KUKA KRL program: MyProgram_321().src

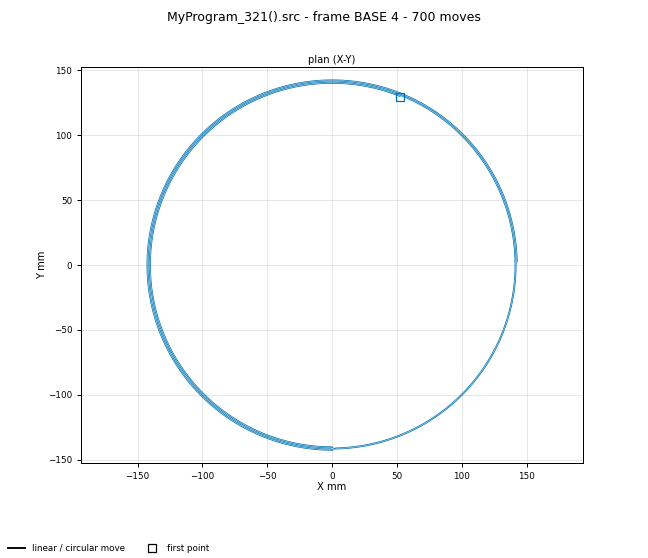
[picture p0: tool path of MyProgram_321().src in frame BASE 4, 700 of 700 moves have a stored position in this frame; points joined in program order, loops and branches not executed]
&ACCESS RVP
&REL 1
&PARAM TEMPLATE = C:\KRC\Roboter\Template\vorgabe
&PARAM EDITMASK = *
DEF MyProgram_321()
; ---- Setting reference (Base) ----
$BASE = BASE_DATA[4]

; --------------------------
; ---- Setting tool (TCP) ----
$TOOL = TOOL_DATA[3]
; --------------------------

$VEL.CP = VEL_APROX_PRINT
Startdeposition()
$VEL.CP = VEL_PRINT
LIN {X 52.4784,Y 129.8657,Z 185,A 69.2762,B 3.164,C 0.0488,E1 3.2265,E2 384.2323} C_DIS
LIN {X 48.957,Y 131.2338,Z 185,A 70.7687,B 3.164,C 0.0476,E1 3.2226,E2 382.7467} C_DIS
LIN {X 45.9323,Y 132.3228,Z 185,A 72.6988,B 3.1641,C 0.0412,E1 3.2173,E2 380.7393} C_DIS
LIN {X 40.835,Y 133.9837,Z 185,A 74.2685,B 3.1641,C 0.0442,E1 3.2133,E2 379.2487} C_DIS
LIN {X 36.7501,Y 135.1629,Z 185,A 76.0213,B 3.1641,C 0.0425,E1 3.2086,E2 377.4947} C_DIS
LIN {X 30.8856,Y 136.621,Z 185,A 78.4846,B 3.1641,C 0.0407,E1 3.2019,E2 375.0331} C_DIS
LIN {X 26.715,Y 137.4977,Z 185,A 80.1371,B 3.1641,C 0.0402,E1 3.1974,E2 373.3925} C_DIS
LIN {X 23.202,Y 138.1334,Z 185,A 81.6304,B 3.1641,C 0.0391,E1 3.1933,E2 371.8956} C_DIS
LIN {X 18.8029,Y 138.802,Z 185,A 83.4433,B 3.1641,C 0.0382,E1 3.1883,E2 370.0842} C_DIS
LIN {X 14.8755,Y 139.2764,Z 185,A 85,B 3.1641,C 0.038,E1 3.184,E2 368.5357} C_DIS
LIN {X 10.3375,Y 139.6866,Z 185,A 86.808,B 3.1641,C 0.0378,E1 3.1789,E2 366.7354} C_DIS
LIN {X 6.929,Y 139.8971,Z 185,A 88.2055,B 3.1641,C 0.0374,E1 3.175,E2 365.3384} C_DIS
LIN {X 2.7761,Y 140.0418,Z 185,A 89.9222,B 3.1641,C 0.0369,E1 3.1702,E2 363.6202} C_DIS
LIN {X -0.9212,Y 140.0657,Z 185,A 91.4585,B 3.1641,C 0.0366,E1 3.1659,E2 362.0816} C_DIS
LIN {X -5.0294,Y 139.9789,Z 185,A 93.0218,B 3.1641,C 0.0373,E1 3.1616,E2 360.5337} C_DIS
LIN {X -7.7827,Y 139.854,Z 185,A 94.1739,B 3.1641,C 0.0372,E1 3.1584,E2 359.379} C_DIS
LIN {X -12.7261,Y 139.4908,Z 185,A 96.4291,B 3.1641,C 0.0359,E1 3.152,E2 357.0964} C_DIS
LIN {X -17.7522,Y 138.9397,Z 185,A 98.302,B 3.1641,C 0.0376,E1 3.1469,E2 355.2489} C_DIS
LIN {X -25.5966,Y 137.7115,Z 185,A 101.6051,B 3.1641,C 0.0384,E1 3.1378,E2 351.9408} C_DIS
LIN {X -29.2647,Y 136.9774,Z 185,A 103.1398,B 3.1641,C 0.039,E1 3.1336,E2 350.4064} C_DIS
LIN {X -32.7165,Y 136.1938,Z 185,A 104.5303,B 3.1641,C 0.0402,E1 3.1298,E2 349.0238} C_DIS
LIN {X -38.5919,Y 134.6492,Z 185,A 107.2007,B 3.1641,C 0.0406,E1 3.1225,E2 346.3318} C_DIS
LIN {X -42.3059,Y 133.5269,Z 185,A 108.7143,B 3.1641,C 0.0422,E1 3.1185,E2 344.8283} C_DIS
LIN {X -45.7058,Y 132.4013,Z 185,A 110.8534,B 3.1641,C 0.0393,E1 3.1127,E2 342.6055} C_DIS
LIN {X -50.7293,Y 130.5589,Z 185,A 112.1604,B 3.1641,C 0.0465,E1 3.1095,E2 341.4104} C_DIS
LIN {X -55.3027,Y 128.6887,Z 185,A 114.4201,B 3.1641,C 0.0471,E1 3.1036,E2 339.1224} C_DIS
LIN {X -58.8401,Y 127.1098,Z 185,A 116.8006,B 3.1641,C 0.0443,E1 3.0973,E2 336.6429} C_DIS
LIN {X -63.9664,Y 124.6097,Z 185,A 118.5759,B 3.164,C 0.0502,E1 3.0931,E2 334.9394} C_DIS
LIN {X -68.2739,Y 122.3048,Z 185,A 120.4705,B 3.164,C 0.0533,E1 3.0885,E2 333.0593} C_DIS
LIN {X -74.5284,Y 118.5969,Z 185,A 123.556,B 3.1639,C 0.0567,E1 3.0811,E2 329.962} C_DIS
LIN {X -78.8304,Y 115.7823,Z 185,A 125.8043,B 3.1639,C 0.0591,E1 3.0758,E2 327.697} C_DIS
LIN {X -81.5053,Y 113.9145,Z 185,A 127.0864,B 3.1638,C 0.0614,E1 3.0729,E2 326.4225} C_DIS
LIN {X -85.6732,Y 110.8141,Z 185,A 129.3317,B 3.1638,C 0.0643,E1 3.0678,E2 324.1635} C_DIS
LIN {X -89.0689,Y 108.104,Z 185,A 131.1966,B 3.1637,C 0.0669,E1 3.0638,E2 322.289} C_DIS
LIN {X -92.6109,Y 105.0851,Z 185,A 133.0845,B 3.1636,C 0.0703,E1 3.0598,E2 320.4045} C_DIS
LIN {X -96.3972,Y 101.6236,Z 185,A 135.298,B 3.1636,C 0.0737,E1 3.0552,E2 318.1781} C_DIS
LIN {X -99.6635,Y 98.4224,Z 185,A 137.2316,B 3.1634,C 0.077,E1 3.0514,E2 316.238} C_DIS
LIN {X -103.1167,Y 94.7975,Z 185,A 140.1431,B 3.1634,C 0.077,E1 3.0457,E2 313.218} C_DIS
LIN {X -107.4445,Y 89.8629,Z 185,A 142.3606,B 3.1632,C 0.0849,E1 3.0418,E2 311.0625} C_DIS
LIN {X -109.699,Y 87.0963,Z 185,A 143.6185,B 3.1632,C 0.0889,E1 3.0396,E2 309.8313} C_DIS
LIN {X -112.4619,Y 83.4983,Z 185,A 145.5483,B 3.163,C 0.0927,E1 3.0364,E2 307.8936} C_DIS
LIN {X -115.0668,Y 79.8704,Z 185,A 147.4654,B 3.1629,C 0.0965,E1 3.0333,E2 305.9664} C_DIS
LIN {X -119.0581,Y 73.7892,Z 185,A 150.54,B 3.1627,C 0.103,E1 3.0286,E2 302.8815} C_DIS
LIN {X -120.8334,Y 70.8445,Z 185,A 151.945,B 3.1626,C 0.1064,E1 3.0266,E2 301.4779} C_DIS
LIN {X -122.9736,Y 67.0605,Z 185,A 153.8444,B 3.1625,C 0.1102,E1 3.024,E2 299.5644} C_DIS
LIN {X -124.5451,Y 64.0933,Z 185,A 155.2767,B 3.1623,C 0.1133,E1 3.0222,E2 298.1256} C_DIS
LIN {X -126.2478,Y 60.6684,Z 185,A 156.8353,B 3.1622,C 0.1173,E1 3.0203,E2 296.569} C_DIS
LIN {X -127.7708,Y 57.391,Z 185,A 158.3489,B 3.1621,C 0.1209,E1 3.0185,E2 295.0519} C_DIS
LIN {X -129.0883,Y 54.3641,Z 185,A 159.7372,B 3.1619,C 0.1242,E1 3.017,E2 293.6598} C_DIS
LIN {X -130.466,Y 50.9682,Z 185,A 161.2824,B 3.1618,C 0.128,E1 3.0154,E2 292.1099} C_DIS
LIN {X -131.5729,Y 48.0416,Z 185,A 162.7467,B 3.1617,C 0.1306,E1 3.0139,E2 290.623} C_DIS
LIN {X -132.8162,Y 44.4861,Z 185,A 164.1953,B 3.1615,C 0.1351,E1 3.0126,E2 289.1873} C_DIS
LIN {X -133.829,Y 41.3404,Z 185,A 165.7134,B 3.1614,C 0.138,E1 3.0113,E2 287.6488} C_DIS
LIN {X -134.846,Y 37.8905,Z 185,A 167.2223,B 3.1612,C 0.1418,E1 3.0102,E2 286.1362} C_DIS
LIN {X -135.7606,Y 34.47,Z 185,A 168.7521,B 3.161,C 0.1454,E1 3.0091,E2 284.597} C_DIS
LIN {X -136.419,Y 31.77,Z 185,A 170.3272,B 3.161,C 0.1468,E1 3.0081,E2 282.966} C_DIS
LIN {X -137.2133,Y 28.1373,Z 185,A 171.504,B 3.1607,C 0.1524,E1 3.0074,E2 281.835} C_DIS
LIN {X -137.9006,Y 24.5479,Z 185,A 173.1137,B 3.1605,C 0.156,E1 3.0066,E2 280.2115} C_DIS
LIN {X -138.8499,Y 18.4371,Z 185,A 175.763,B 3.1602,C 0.1626,E1 3.0055,E2 277.5486} C_DIS
LIN {X -139.6415,Y 10.9549,Z 185,A 178.9229,B 3.1598,C 0.1709,E1 3.0046,E2 274.3803} C_DIS
LIN {X -140.0189,Y 3.7363,Z 185,A -178.036,B 3.1593,C 0.1789,E1 3.0042,E2 271.3304} C_DIS
LIN {X -140.055,Y -1.9821,Z 185,A -175.4265,B 3.159,C 0.1844,E1 3.0042,E2 268.6873} C_DIS
LIN {X -139.5897,Y -11.5732,Z 185,A -170.7123,B 3.1585,C 0.1922,E1 3.0051,E2 263.8721} C_DIS
LIN {X -139.065,Y -16.7372,Z 185,A -169.1009,B 3.158,C 0.2003,E1 3.0055,E2 262.3295} C_DIS
LIN {X -138.623,Y -20.0725,Z 185,A -166.986,B 3.158,C 0.2011,E1 3.0065,E2 260.1178} C_DIS
LIN {X -137.7112,Y -25.5985,Z 185,A -165.226,B 3.1574,C 0.2096,E1 3.0073,E2 258.4296} C_DIS
LIN {X -136.9555,Y -29.3659,Z 185,A -163.6667,B 3.1571,C 0.214,E1 3.0082,E2 256.8728} C_DIS
LIN {X -136.23,Y -32.5664,Z 185,A -162.2465,B 3.1569,C 0.2173,E1 3.0091,E2 255.443} C_DIS
LIN {X -135.335,Y -36.1048,Z 185,A -160.6663,B 3.1567,C 0.221,E1 3.0102,E2 253.8521} C_DIS
LIN {X -134.1672,Y -40.2355,Z 185,A -158.7607,B 3.1564,C 0.2251,E1 3.0117,E2 251.9276} C_DIS
LIN {X -133.023,Y -43.8651,Z 185,A -157.2747,B 3.156,C 0.2295,E1 3.013,E2 250.4517} C_DIS
LIN {X -132.1127,Y -46.5382,Z 185,A -155.6379,B 3.156,C 0.2305,E1 3.0145,E2 248.7514} C_DIS
LIN {X -130.8306,Y -50.0258,Z 185,A -154.2107,B 3.1557,C 0.2348,E1 3.0159,E2 247.3372} C_DIS
LIN {X -128.9154,Y -54.7767,Z 185,A -152.0339,B 3.1553,C 0.2398,E1 3.0183,E2 245.1505} C_DIS
LIN {X -127.1672,Y -58.7159,Z 185,A -150.4445,B 3.1549,C 0.2451,E1 3.0201,E2 243.5849} C_DIS
LIN {X -125.7276,Y -61.7389,Z 185,A -148.97,B 3.1546,C 0.248,E1 3.0219,E2 242.097} C_DIS
LIN {X -124.2342,Y -64.6926,Z 185,A -147.7027,B 3.1543,C 0.2517,E1 3.0235,E2 240.8418} C_DIS
LIN {X -122.1164,Y -68.6088,Z 185,A -145.3764,B 3.1542,C 0.2538,E1 3.0267,E2 238.4485} C_DIS
LIN {X -120.4117,Y -71.5588,Z 185,A -144.1967,B 3.1538,C 0.2581,E1 3.0284,E2 237.2981} C_DIS
LIN {X -118.7534,Y -74.2785,Z 185,A -142.757,B 3.1536,C 0.2605,E1 3.0305,E2 235.8404} C_DIS
LIN {X -116.2436,Y -78.1488,Z 185,A -140.8018,B 3.1533,C 0.2645,E1 3.0335,E2 233.8766} C_DIS
LIN {X -113.711,Y -81.7899,Z 185,A -137.9116,B 3.1534,C 0.2632,E1 3.0386,E2 230.8409} C_DIS
LIN {X -109.0174,Y -87.9479,Z 185,A -135.6805,B 3.1524,C 0.2747,E1 3.0422,E2 228.738} C_DIS
LIN {X -106.4108,Y -91.0853,Z 185,A -133.6686,B 3.1523,C 0.2764,E1 3.0459,E2 226.6799} C_DIS
LIN {X -103.9814,Y -93.8489,Z 185,A -132.3653,B 3.1519,C 0.2805,E1 3.0483,E2 225.4043} C_DIS
LIN {X -100.9241,Y -97.1294,Z 185,A -130.5328,B 3.1516,C 0.2841,E1 3.0518,E2 223.5724} C_DIS
LIN {X -95.0469,Y -102.8874,Z 185,A -126.9885,B 3.1511,C 0.2894,E1 3.059,E2 220.0045} C_DIS
LIN {X -92.8343,Y -104.8876,Z 185,A -125.606,B 3.1511,C 0.2906,E1 3.0619,E2 218.6} C_DIS
LIN {X -88.7193,Y -108.3906,Z 185,A -123.4952,B 3.1506,C 0.2949,E1 3.0664,E2 216.5029} C_DIS
LIN {X -85.3042,Y -111.0985,Z 185,A -121.5078,B 3.1504,C 0.2967,E1 3.0708,E2 214.4877} C_DIS
LIN {X -79.2766,Y -115.4766,Z 185,A -118.5366,B 3.15,C 0.3017,E1 3.0776,E2 211.527} C_DIS
LIN {X -75.52,Y -117.9676,Z 185,A -116.6646,B 3.1497,C 0.3042,E1 3.082,E2 209.6511} C_DIS
LIN {X -71.562,Y -120.4098,Z 185,A -114.7317,B 3.1495,C 0.3065,E1 3.0866,E2 207.7139} C_DIS
LIN {X -67.6087,Y -122.6734,Z 185,A -112.7489,B 3.1493,C 0.3081,E1 3.0915,E2 205.7146} C_DIS
LIN {X -61.8436,Y -125.6759,Z 185,A -110.203,B 3.149,C 0.3118,E1 3.0978,E2 203.184} C_DIS
LIN {X -58.0218,Y -127.4882,Z 185,A -108.2284,B 3.149,C 0.3121,E1 3.1029,E2 201.1757} C_DIS
LIN {X -53.8818,Y -129.2897,Z 185,A -106.5178,B 3.1487,C 0.3147,E1 3.1072,E2 199.4833} C_DIS
LIN {X -49.9004,Y -130.8805,Z 185,A -104.7913,B 3.1485,C 0.3165,E1 3.1117,E2 197.7604} C_DIS
LIN {X -43.8112,Y -133.0409,Z 185,A -102.0488,B 3.1484,C 0.3178,E1 3.119,E2 195.0037} C_DIS
LIN {X -39.8106,Y -134.2924,Z 185,A -100.3133,B 3.1483,C 0.3188,E1 3.1236,E2 193.2649} C_DIS
LIN {X -33.7193,Y -135.9511,Z 185,A -97.4739,B 3.1483,C 0.3185,E1 3.1314,E2 190.3895} C_DIS
LIN {X -30.5364,Y -136.7008,Z 185,A -96.3207,B 3.1481,C 0.3204,E1 3.1345,E2 189.2612} C_DIS
LIN {X -26.4818,Y -137.5423,Z 185,A -94.5632,B 3.1481,C 0.3206,E1 3.1393,E2 187.4943} C_DIS
LIN {X -21.6911,Y -138.3789,Z 185,A -92.6937,B 3.148,C 0.3221,E1 3.1445,E2 185.6406} C_DIS
LIN {X -18.1946,Y -138.8817,Z 185,A -91.296,B 3.1479,C 0.3227,E1 3.1483,E2 184.2489} C_DIS
LIN {X -15.1048,Y -139.2517,Z 185,A -90.0586,B 3.1479,C 0.3232,E1 3.1517,E2 183.0159} C_DIS
LIN {X -11.7315,Y -139.5764,Z 185,A -88.5818,B 3.1479,C 0.3226,E1 3.1559,E2 181.5261} C_DIS
LIN {X -7.5843,Y -139.8642,Z 185,A -86.8184,B 3.1479,C 0.3222,E1 3.1608,E2 179.7533} C_DIS
LIN {X -4.0287,Y -140.0107,Z 185,A -85.4305,B 3.1479,C 0.3226,E1 3.1647,E2 178.3741} C_DIS
LIN {X -0.2852,Y -140.0692,Z 185,A -83.8235,B 3.1479,C 0.3218,E1 3.1692,E2 176.756} C_DIS
LIN {X -0.2852,Y -140.0692,Z 185,A -83.8235,B 3.1479,C 0.3218,E1 3.1692,E2 176.756} C_DIS
Enddeposition()
LIN {X 0.9983,Y -140.9641,Z 185,A -83.429,B 3.1812,C 0.3256,E1 3.2037,E2 176.4} C_DIS
Startdeposition()
$VEL.CP = VEL_PRINT
LIN {X -2.7363,Y -140.9428,Z 185,A -85.6556,B 3.1806,C 0.3313,E1 3.1972,E2 178.725} C_DIS
LIN {X -7.0932,Y -140.7902,Z 185,A -87.2838,B 3.1807,C 0.3303,E1 3.1927,E2 180.3343} C_DIS
LIN {X -10.3887,Y -140.5854,Z 185,A -88.6415,B 3.1807,C 0.3303,E1 3.1889,E2 181.6947} C_DIS
LIN {X -13.9414,Y -140.2784,Z 185,A -90.0893,B 3.1807,C 0.3303,E1 3.1849,E2 183.1429} C_DIS
LIN {X -17.9054,Y -139.8275,Z 185,A -91.7624,B 3.1807,C 0.3303,E1 3.1802,E2 184.8237} C_DIS
LIN {X -21.5636,Y -139.3095,Z 185,A -93.2532,B 3.1807,C 0.3299,E1 3.1761,E2 186.3135} C_DIS
LIN {X -25.4241,Y -138.6582,Z 185,A -94.807,B 3.1809,C 0.3291,E1 3.1718,E2 187.8628} C_DIS
LIN {X -28.2372,Y -138.1115,Z 185,A -96.0268,B 3.1809,C 0.3291,E1 3.1685,E2 189.0905} C_DIS
LIN {X -31.6567,Y -137.3683,Z 185,A -97.4512,B 3.1809,C 0.3284,E1 3.1646,E2 190.5156} C_DIS
LIN {X -35.5194,Y -136.4223,Z 185,A -99.0391,B 3.181,C 0.3273,E1 3.1603,E2 192.1002} C_DIS
LIN {X -39.2475,Y -135.3952,Z 185,A -100.4748,B 3.1812,C 0.3255,E1 3.1565,E2 193.5176} C_DIS
LIN {X -42.1974,Y -134.5065,Z 185,A -102.3715,B 3.1809,C 0.329,E1 3.1512,E2 195.5026} C_DIS
LIN {X -46.0988,Y -133.2178,Z 185,A -103.7302,B 3.1812,C 0.3256,E1 3.1477,E2 196.8193} C_DIS
LIN {X -49.909,Y -131.8385,Z 185,A -105.2692,B 3.1814,C 0.3236,E1 3.1437,E2 198.344} C_DIS
LIN {X -53.6025,Y -130.3819,Z 185,A -107.027,B 3.1814,C 0.323,E1 3.1391,E2 200.1218} C_DIS
LIN {X -57.8864,Y -128.5353,Z 185,A -108.8479,B 3.1817,C 0.3207,E1 3.1344,E2 201.9327} C_DIS
LIN {X -61.157,Y -127.012,Z 185,A -110.3275,B 3.1819,C 0.3192,E1 3.1307,E2 203.4143} C_DIS
LIN {X -64.5951,Y -125.2997,Z 185,A -112.3787,B 3.1817,C 0.3205,E1 3.1254,E2 205.5322} C_DIS
LIN {X -68.3459,Y -123.2941,Z 185,A -113.6031,B 3.1823,C 0.3153,E1 3.1226,E2 206.6883} C_DIS
LIN {X -71.6589,Y -121.3989,Z 185,A -115.3609,B 3.1823,C 0.3145,E1 3.1183,E2 208.4744} C_DIS
LIN {X -75.6376,Y -118.9611,Z 185,A -117.1095,B 3.1827,C 0.3111,E1 3.1142,E2 210.2029} C_DIS
LIN {X -78.4609,Y -117.1177,Z 185,A -118.6732,B 3.1827,C 0.3103,E1 3.1104,E2 211.793} C_DIS
LIN {X -82.0881,Y -114.6044,Z 185,A -121.0227,B 3.1827,C 0.3108,E1 3.1049,E2 214.2175} C_DIS
LIN {X -86.0238,Y -111.6812,Z 185,A -122.5769,B 3.1832,C 0.3051,E1 3.1016,E2 215.7126} C_DIS
LIN {X -89.5299,Y -108.8907,Z 185,A -124.465,B 3.1835,C 0.3025,E1 3.0975,E2 217.6096} C_DIS
LIN {X -93.7841,Y -105.2486,Z 185,A -126.6118,B 3.1839,C 0.2978,E1 3.093,E2 219.7387} C_DIS
LIN {X -99.8151,Y -99.5471,Z 185,A -130.1775,B 3.1844,C 0.2926,E1 3.0857,E2 223.3301} C_DIS
LIN {X -102.6757,Y -96.5937,Z 185,A -131.8436,B 3.1847,C 0.2893,E1 3.0825,E2 224.9953} C_DIS
LIN {X -105.2598,Y -93.7717,Z 185,A -133.998,B 3.1847,C 0.2893,E1 3.0783,E2 227.2299} C_DIS
LIN {X -108.0974,Y -90.4853,Z 185,A -135.2848,B 3.1853,C 0.2832,E1 3.0761,E2 228.4523} C_DIS
LIN {X -114.3775,Y -82.4048,Z 185,A -139.6464,B 3.186,C 0.2753,E1 3.0687,E2 232.8402} C_DIS
LIN {X -116.6269,Y -79.1884,Z 185,A -141.4084,B 3.1862,C 0.2724,E1 3.0658,E2 234.6241} C_DIS
LIN {X -119.3393,Y -75.0387,Z 185,A -143.3993,B 3.1866,C 0.2677,E1 3.0628,E2 236.6111} C_DIS
LIN {X -121.3686,Y -71.7104,Z 185,A -145.1358,B 3.1869,C 0.2647,E1 3.0603,E2 238.3674} C_DIS
LIN {X -124.4839,Y -66.1534,Z 185,A -147.6638,B 3.1874,C 0.2581,E1 3.0569,E2 240.8863} C_DIS
LIN {X -125.7613,Y -63.6884,Z 185,A -148.9129,B 3.1876,C 0.2559,E1 3.0553,E2 242.151} C_DIS
LIN {X -127.3943,Y -60.3567,Z 185,A -150.5507,B 3.1878,C 0.2527,E1 3.0533,E2 243.8054} C_DIS
LIN {X -129.5032,Y -55.687,Z 185,A -152.6726,B 3.1882,C 0.2476,E1 3.0509,E2 245.9317} C_DIS
LIN {X -130.9413,Y -52.2179,Z 185,A -154.2465,B 3.1885,C 0.2439,E1 3.0492,E2 247.5112} C_DIS
LIN {X -132.9886,Y -46.76,Z 185,A -156.6139,B 3.189,C 0.2377,E1 3.0469,E2 249.8773} C_DIS
LIN {X -134.3341,Y -42.7369,Z 185,A -158.5318,B 3.1893,C 0.234,E1 3.0452,E2 251.82} C_DIS
LIN {X -135.3324,Y -39.462,Z 185,A -159.9598,B 3.1895,C 0.2304,E1 3.0441,E2 253.252} C_DIS
LIN {X -136.2157,Y -36.2956,Z 185,A -161.3695,B 3.1897,C 0.2271,E1 3.043,E2 254.6708} C_DIS
LIN {X -137.102,Y -32.7903,Z 185,A -162.8528,B 3.19,C 0.2232,E1 3.042,E2 256.1552} C_DIS
LIN {X -137.8714,Y -29.3893,Z 185,A -164.4735,B 3.1902,C 0.2201,E1 3.0411,E2 257.8018} C_DIS
LIN {X -139.5391,Y -20.0246,Z 185,A -168.412,B 3.1909,C 0.2098,E1 3.0392,E2 261.7476} C_DIS
LIN {X -140.4751,Y -11.7867,Z 185,A -171.824,B 3.1915,C 0.2005,E1 3.0382,E2 265.1632} C_DIS
LIN {X -140.8473,Y -5.8611,Z 185,A -174.4728,B 3.1919,C 0.1947,E1 3.0378,E2 267.8415} C_DIS
LIN {X -140.9513,Y -2.2221,Z 185,A -175.9858,B 3.1921,C 0.1907,E1 3.0376,E2 269.3578} C_DIS
LIN {X -140.9638,Y 1.3399,Z 185,A -177.8771,B 3.1923,C 0.1884,E1 3.0376,E2 271.3057} C_DIS
LIN {X -140.8872,Y 4.8334,Z 185,A -179.5218,B 3.1924,C 0.1853,E1 3.0378,E2 272.9784} C_DIS
LIN {X -140.674,Y 9.122,Z 185,A 179.2569,B 3.1928,C 0.1783,E1 3.038,E2 274.1309} C_DIS
LIN {X -140.464,Y 11.9179,Z 185,A 177.9635,B 3.193,C 0.1757,E1 3.0383,E2 275.4434} C_DIS
LIN {X -140.1533,Y 15.1396,Z 185,A 176.524,B 3.1932,C 0.1725,E1 3.0387,E2 276.8981} C_DIS
LIN {X -139.7794,Y 18.2723,Z 185,A 174.5569,B 3.1932,C 0.1717,E1 3.0395,E2 278.9521} C_DIS
LIN {X -138.9929,Y 23.5205,Z 185,A 173.3088,B 3.1937,C 0.162,E1 3.04,E2 280.082} C_DIS
LIN {X -138.5135,Y 26.1954,Z 185,A 171.5293,B 3.1937,C 0.1617,E1 3.0409,E2 281.9477} C_DIS
LIN {X -137.8737,Y 29.377,Z 185,A 170.3325,B 3.1939,C 0.1576,E1 3.0416,E2 283.1279} C_DIS
LIN {X -137.0328,Y 33.0774,Z 185,A 168.8318,B 3.1941,C 0.1532,E1 3.0426,E2 284.622} C_DIS
LIN {X -136.162,Y 36.4971,Z 185,A 167.314,B 3.1943,C 0.1496,E1 3.0436,E2 286.1495} C_DIS
LIN {X -135.1973,Y 39.9233,Z 185,A 165.8238,B 3.1945,C 0.1459,E1 3.0448,E2 287.6442} C_DIS
LIN {X -134.185,Y 43.2039,Z 185,A 164.3551,B 3.1946,C 0.1424,E1 3.046,E2 289.1213} C_DIS
LIN {X -133.0979,Y 46.4447,Z 185,A 162.8692,B 3.1948,C 0.1391,E1 3.0474,E2 290.6185} C_DIS
LIN {X -131.8137,Y 49.9752,Z 185,A 161.3169,B 3.195,C 0.1352,E1 3.0489,E2 292.1729} C_DIS
LIN {X -130.6022,Y 53.0592,Z 185,A 159.9093,B 3.195,C 0.132,E1 3.0503,E2 293.5872} C_DIS
LIN {X -129.2467,Y 56.2802,Z 185,A 158.4175,B 3.1952,C 0.1286,E1 3.052,E2 295.087} C_DIS
LIN {X -127.7463,Y 59.6084,Z 185,A 156.8715,B 3.1954,C 0.1251,E1 3.0538,E2 296.6398} C_DIS
LIN {X -126.2799,Y 62.6541,Z 185,A 155.4178,B 3.1954,C 0.122,E1 3.0556,E2 298.1025} C_DIS
LIN {X -124.3417,Y 66.422,Z 185,A 153.4721,B 3.1956,C 0.1187,E1 3.0582,E2 300.0753} C_DIS
LIN {X -122.2558,Y 70.1874,Z 185,A 151.729,B 3.1958,C 0.1144,E1 3.0606,E2 301.8163} C_DIS
LIN {X -119.9278,Y 74.0953,Z 185,A 149.7897,B 3.1959,C 0.1104,E1 3.0634,E2 303.7656} C_DIS
LIN {X -115.5588,Y 80.7394,Z 185,A 146.4999,B 3.1962,C 0.1032,E1 3.0685,E2 307.0602} C_DIS
LIN {X -112.9544,Y 84.3443,Z 185,A 144.6514,B 3.1962,C 0.0993,E1 3.0715,E2 308.9125} C_DIS
LIN {X -110.4876,Y 87.551,Z 185,A 142.7743,B 3.1964,C 0.0968,E1 3.0748,E2 310.8176} C_DIS
LIN {X -108.2915,Y 90.2538,Z 185,A 141.3792,B 3.1964,C 0.0937,E1 3.0773,E2 312.2091} C_DIS
LIN {X -103.59,Y 95.6127,Z 185,A 138.418,B 3.1966,C 0.088,E1 3.0828,E2 315.176} C_DIS
LIN {X -100.4352,Y 98.9215,Z 185,A 136.5114,B 3.1966,C 0.0846,E1 3.0865,E2 317.0873} C_DIS
LIN {X -97.3478,Y 101.9609,Z 185,A 134.7,B 3.1968,C 0.0815,E1 3.0902,E2 318.9037} C_DIS
LIN {X -93.3289,Y 105.6519,Z 185,A 132.4126,B 3.1968,C 0.0778,E1 3.0949,E2 321.1982} C_DIS
LIN {X -90.0651,Y 108.4478,Z 185,A 130.6274,B 3.1969,C 0.0749,E1 3.0987,E2 322.9869} C_DIS
LIN {X -86.6725,Y 111.1784,Z 185,A 128.7495,B 3.1969,C 0.0725,E1 3.1029,E2 324.877} C_DIS
LIN {X -81.978,Y 114.6831,Z 185,A 126.6134,B 3.1971,C 0.0674,E1 3.1076,E2 326.9807} C_DIS
LIN {X -79.4091,Y 116.4774,Z 185,A 124.8417,B 3.1971,C 0.0681,E1 3.1118,E2 328.8137} C_DIS
LIN {X -76.7396,Y 118.2525,Z 185,A 123.7604,B 3.1971,C 0.065,E1 3.1143,E2 329.8665} C_DIS
LIN {X -70.1422,Y 122.2816,Z 185,A 120.6227,B 3.1972,C 0.0607,E1 3.1218,E2 333.0016} C_DIS
LIN {X -66.9798,Y 124.042,Z 185,A 118.984,B 3.1972,C 0.0597,E1 3.1259,E2 334.6601} C_DIS
LIN {X -63.6411,Y 125.7854,Z 185,A 116.7901,B 3.1972,C 0.0617,E1 3.1316,E2 336.9349} C_DIS
LIN {X -58.452,Y 128.281,Z 185,A 115.1421,B 3.1973,C 0.0552,E1 3.1355,E2 338.4959} C_DIS
LIN {X -55.3771,Y 129.6372,Z 185,A 113.3711,B 3.1973,C 0.0561,E1 3.1402,E2 340.3163} C_DIS
LIN {X -51.8268,Y 131.098,Z 185,A 111.87,B 3.1973,C 0.0543,E1 3.1441,E2 341.8091} C_DIS
LIN {X -48.7605,Y 132.2687,Z 185,A 110.5377,B 3.1973,C 0.0531,E1 3.1475,E2 343.1403} C_DIS
LIN {X -44.4673,Y 133.7712,Z 185,A 108.8961,B 3.1974,C 0.0504,E1 3.1518,E2 344.7551} C_DIS
LIN {X -40.8547,Y 134.919,Z 185,A 107.2622,B 3.1974,C 0.0498,E1 3.1562,E2 346.3997} C_DIS
LIN {X -35.0004,Y 136.5547,Z 185,A 105.0043,B 3.1974,C 0.0469,E1 3.1622,E2 348.6298} C_DIS
LIN {X -32.1224,Y 137.2619,Z 185,A 102.9401,B 3.1974,C 0.0518,E1 3.1682,E2 350.7995} C_DIS
LIN {X -26.6346,Y 138.4296,Z 185,A 101.2345,B 3.1974,C 0.0471,E1 3.1726,E2 352.433} C_DIS
LIN {X -19.9044,Y 139.5563,Z 185,A 98.5576,B 3.1974,C 0.0455,E1 3.18,E2 355.0966} C_DIS
LIN {X -16.1174,Y 140.0454,Z 185,A 96.98,B 3.1974,C 0.0453,E1 3.1844,E2 356.6766} C_DIS
LIN {X -12.1432,Y 140.445,Z 185,A 94.7167,B 3.1974,C 0.0494,E1 3.1909,E2 359.018} C_DIS
LIN {X -6.6681,Y 140.8116,Z 185,A 93.1898,B 3.1975,C 0.0445,E1 3.1949,E2 360.4572} C_DIS
LIN {X -2.9181,Y 140.9398,Z 185,A 91.5624,B 3.1975,C 0.0453,E1 3.1995,E2 362.0967} C_DIS
LIN {X 0.8338,Y 140.9664,Z 185,A 90.057,B 3.1975,C 0.0453,E1 3.2037,E2 363.599} C_DIS
LIN {X 5.436,Y 140.8639,Z 185,A 88.2301,B 3.1975,C 0.0453,E1 3.2088,E2 365.4197} C_DIS
LIN {X 9.5085,Y 140.6497,Z 185,A 86.4742,B 3.1975,C 0.0466,E1 3.2137,E2 367.1872} C_DIS
LIN {X 13.4404,Y 140.3265,Z 185,A 85.0006,B 3.1975,C 0.0462,E1 3.2178,E2 368.644} C_DIS
LIN {X 17.0733,Y 139.9314,Z 185,A 83.4555,B 3.1975,C 0.0473,E1 3.2221,E2 370.196} C_DIS
LIN {X 22.7151,Y 139.1273,Z 185,A 81.3664,B 3.1975,C 0.0468,E1 3.2278,E2 372.2562} C_DIS
LIN {X 26.5686,Y 138.4422,Z 185,A 79.6439,B 3.1975,C 0.0488,E1 3.2325,E2 373.9946} C_DIS
LIN {X 30.285,Y 137.678,Z 185,A 78.1315,B 3.1975,C 0.0496,E1 3.2367,E2 375.5028} C_DIS
LIN {X 32.9583,Y 137.0615,Z 185,A 76.7749,B 3.1974,C 0.0524,E1 3.2404,E2 376.8891} C_DIS
LIN {X 37.2544,Y 135.9586,Z 185,A 75.1382,B 3.1974,C 0.0526,E1 3.2448,E2 378.5048} C_DIS
LIN {X 43.2924,Y 134.1567,Z 185,A 72.4081,B 3.1974,C 0.0563,E1 3.2521,E2 381.2553} C_DIS
LIN {X 46.6543,Y 133.0252,Z 185,A 71.3248,B 3.1974,C 0.0549,E1 3.2549,E2 382.2937} C_DIS
LIN {X 49.8012,Y 131.8789,Z 185,A 69.9548,B 3.1974,C 0.0564,E1 3.2585,E2 383.6647} C_DIS
LIN {X 53.0027,Y 130.6249,Z 185,A 68.5929,B 3.1973,C 0.0577,E1 3.262,E2 385.0218} C_DIS
LIN {X 56.4984,Y 129.1524,Z 185,A 67.1017,B 3.1973,C 0.0592,E1 3.2658,E2 386.5065} C_DIS
LIN {X 59.3563,Y 127.8628,Z 185,A 65.8218,B 3.1973,C 0.0608,E1 3.2691,E2 387.7869} C_DIS
LIN {X 62.3849,Y 126.4127,Z 185,A 64.1647,B 3.1972,C 0.0651,E1 3.2733,E2 389.4803} C_DIS
LIN {X 65.6133,Y 124.7675,Z 185,A 63.3014,B 3.1972,C 0.062,E1 3.2753,E2 390.2673} C_DIS
LIN {X 68.6292,Y 123.1373,Z 185,A 61.5893,B 3.1972,C 0.0667,E1 3.2796,E2 392.0195} C_DIS
LIN {X 72.5892,Y 120.8453,Z 185,A 59.7716,B 3.1971,C 0.0692,E1 3.2839,E2 393.8318} C_DIS
LIN {X 76.4538,Y 118.438,Z 185,A 58.0087,B 3.1971,C 0.0713,E1 3.2881,E2 395.5837} C_DIS
LIN {X 80.1308,Y 115.9821,Z 185,A 55.9753,B 3.1969,C 0.0764,E1 3.2928,E2 397.6467} C_DIS
LIN {X 83.1496,Y 113.8372,Z 185,A 54.7503,B 3.1969,C 0.0765,E1 3.2955,E2 398.8366} C_DIS
LIN {X 86.7521,Y 111.1164,Z 185,A 52.9553,B 3.1969,C 0.0794,E1 3.2995,E2 400.6267} C_DIS
LIN {X 90.4738,Y 108.107,Z 185,A 51.0777,B 3.1968,C 0.0824,E1 3.3035,E2 402.4958} C_DIS
LIN {X 93.9423,Y 105.1069,Z 185,A 48.9028,B 3.1966,C 0.0889,E1 3.3082,E2 404.7101} C_DIS
LIN {X 97.2087,Y 102.0938,Z 185,A 47.5313,B 3.1966,C 0.0885,E1 3.3108,E2 406.0271} C_DIS
LIN {X 100.4314,Y 98.9254,Z 185,A 45.7274,B 3.1965,C 0.0919,E1 3.3144,E2 407.8271} C_DIS
LIN {X 103.6394,Y 95.559,Z 185,A 43.9244,B 3.1965,C 0.0951,E1 3.3178,E2 409.6194} C_DIS
LIN {X 106.4369,Y 92.4332,Z 185,A 42.2578,B 3.1963,C 0.0984,E1 3.3209,E2 411.2814} C_DIS
LIN {X 109.4417,Y 88.8555,Z 185,A 40.1267,B 3.1961,C 0.1048,E1 3.3247,E2 413.4425} C_DIS
LIN {X 111.9295,Y 85.6994,Z 185,A 38.9547,B 3.1961,C 0.1041,E1 3.3266,E2 414.5563} C_DIS
LIN {X 114.3921,Y 82.3846,Z 185,A 37.238,B 3.196,C 0.1083,E1 3.3295,E2 416.2783} C_DIS
LIN {X 116.9708,Y 78.6804,Z 185,A 35.4459,B 3.1958,C 0.1122,E1 3.3323,E2 418.0655} C_DIS
LIN {X 119.4952,Y 74.7906,Z 185,A 33.6429,B 3.1958,C 0.116,E1 3.335,E2 419.8587} C_DIS
LIN {X 121.8391,Y 70.9079,Z 185,A 31.8883,B 3.1956,C 0.1196,E1 3.3375,E2 421.6025} C_DIS
LIN {X 124.0255,Y 67.0105,Z 185,A 30.1224,B 3.1954,C 0.1236,E1 3.3398,E2 423.3627} C_DIS
LIN {X 125.9252,Y 63.3664,Z 185,A 28.6297,B 3.1954,C 0.1261,E1 3.3417,E2 424.8331} C_DIS
LIN {X 127.3171,Y 60.5184,Z 185,A 27.3756,B 3.1952,C 0.129,E1 3.3432,E2 426.0832} C_DIS
LIN {X 128.8109,Y 57.2704,Z 185,A 25.9756,B 3.1951,C 0.1323,E1 3.3448,E2 427.477} C_DIS
LIN {X 130.2413,Y 53.9392,Z 185,A 24.5709,B 3.1949,C 0.1354,E1 3.3463,E2 428.8736} C_DIS
LIN {X 131.5259,Y 50.7262,Z 185,A 23.2229,B 3.1949,C 0.1385,E1 3.3477,E2 430.2146} C_DIS
LIN {X 132.7987,Y 47.2957,Z 185,A 21.8193,B 3.1947,C 0.1416,E1 3.3491,E2 431.6081} C_DIS
LIN {X 133.8517,Y 44.2257,Z 185,A 20.5108,B 3.1945,C 0.1451,E1 3.3502,E2 432.9158} C_DIS
LIN {X 135.1163,Y 40.2002,Z 185,A 18.2414,B 3.194,C 0.1554,E1 3.3521,E2 435.2575} C_DIS
LIN {X 136.5633,Y 34.9664,Z 185,A 16.951,B 3.1942,C 0.152,E1 3.3529,E2 436.4306} C_DIS
LIN {X 138.2482,Y 27.5657,Z 185,A 13.2573,B 3.1935,C 0.1668,E1 3.3552,E2 440.205} C_DIS
LIN {X 139.134,Y 22.6747,Z 185,A 11.9064,B 3.1935,C 0.1655,E1 3.3558,E2 441.4703} C_DIS
LIN {X 139.5856,Y 19.6991,Z 185,A 10.7349,B 3.1934,C 0.1684,E1 3.3562,E2 442.6358} C_DIS
LIN {X 139.9926,Y 16.5599,Z 185,A 9.477,B 3.1932,C 0.1717,E1 3.3567,E2 443.8906} C_DIS
LIN {X 140.4118,Y 12.5358,Z 185,A 7.7926,B 3.1929,C 0.1767,E1 3.3571,E2 445.5814} C_DIS
LIN {X 140.7095,Y 8.5459,Z 185,A 6.3285,B 3.1928,C 0.1796,E1 3.3574,E2 447.0252} C_DIS
LIN {X 140.8948,Y 4.6218,Z 185,A 4.7103,B 3.1925,C 0.1843,E1 3.3576,E2 448.6473} C_DIS
LIN {X 140.969,Y 0.5279,Z 185,A 3.2581,B 3.1924,C 0.1868,E1 3.3576,E2 450.0728} C_DIS
LIN {X 140.9432,Y -2.7135,Z 185,A 1.8732,B 3.1921,C 0.1912,E1 3.3576,E2 451.4673} C_DIS
LIN {X 140.7971,Y -6.9562,Z 185,A 0.2936,B 3.1919,C 0.1946,E1 3.3574,E2 453.0289} C_DIS
LIN {X 140.5573,Y -10.7744,Z 185,A -1.299,B 3.1916,C 0.1993,E1 3.3571,E2 454.6275} C_DIS
LIN {X 140.1691,Y -14.9935,Z 185,A -2.8679,B 3.1914,C 0.2026,E1 3.3567,E2 456.1774} C_DIS
LIN {X 139.6796,Y -19.0337,Z 185,A -4.6063,B 3.191,C 0.2081,E1 3.356,E2 457.9281} C_DIS
LIN {X 138.9806,Y -23.5943,Z 185,A -6.2157,B 3.1909,C 0.2105,E1 3.3553,E2 459.5037} C_DIS
LIN {X 138.3132,Y -27.2432,Z 185,A -8.002,B 3.1904,C 0.2176,E1 3.3544,E2 461.3281} C_DIS
LIN {X 137.5544,Y -30.8416,Z 185,A -8.9937,B 3.1904,C 0.2165,E1 3.3538,E2 462.2542} C_DIS
LIN {X 136.5066,Y -35.1886,Z 185,A -11.0861,B 3.1899,C 0.2244,E1 3.3524,E2 464.3844} C_DIS
LIN {X 135.6723,Y -38.2784,Z 185,A -12.1093,B 3.1899,C 0.225,E1 3.3516,E2 465.3718} C_DIS
LIN {X 133.7529,Y -44.5222,Z 185,A -15.3263,B 3.189,C 0.2381,E1 3.3488,E2 468.6653} C_DIS
LIN {X 131.7673,Y -50.0991,Z 185,A -16.8911,B 3.1891,C 0.2358,E1 3.3474,E2 470.1204} C_DIS
LIN {X 130.0758,Y -54.3355,Z 185,A -18.6878,B 3.1888,C 0.2401,E1 3.3455,E2 471.9107} C_DIS
LIN {X 128.727,Y -57.458,Z 185,A -20.57,B 3.1881,C 0.2488,E1 3.3433,E2 473.8607} C_DIS
LIN {X 126.6604,Y -61.8827,Z 185,A -21.8332,B 3.1883,C 0.2465,E1 3.3419,E2 475.0292} C_DIS
LIN {X 123.0651,Y -68.7584,Z 185,A -24.9097,B 3.1877,C 0.2538,E1 3.3379,E2 478.0981} C_DIS
LIN {X 121.701,Y -71.1446,Z 185,A -26.1576,B 3.1874,C 0.2578,E1 3.3361,E2 479.3645} C_DIS
LIN {X 119.3687,Y -74.9921,Z 185,A -27.9316,B 3.1871,C 0.2618,E1 3.3335,E2 481.1326} C_DIS
LIN {X 116.6945,Y -79.0885,Z 185,A -29.6986,B 3.1869,C 0.2643,E1 3.3308,E2 482.8714} C_DIS
LIN {X 114.4899,Y -82.2481,Z 185,A -31.6725,B 3.1862,C 0.2721,E1 3.3275,E2 484.9015} C_DIS
LIN {X 111.9738,Y -85.6415,Z 185,A -32.8295,B 3.1864,C 0.2704,E1 3.3257,E2 485.9846} C_DIS
LIN {X 109.5947,Y -88.6659,Z 185,A -34.489,B 3.186,C 0.275,E1 3.3228,E2 487.6583} C_DIS
LIN {X 105.2922,Y -93.734,Z 185,A -37.302,B 3.1854,C 0.282,E1 3.3176,E2 490.4884} C_DIS
LIN {X 102.9784,Y -96.2711,Z 185,A -38.4561,B 3.1854,C 0.2826,E1 3.3155,E2 491.611} C_DIS
LIN {X 97.5667,Y -101.7516,Z 185,A -41.1797,B 3.1851,C 0.2851,E1 3.3102,E2 494.282} C_DIS
LIN {X 91.9653,Y -106.841,Z 185,A -44.8282,B 3.184,C 0.2968,E1 3.3025,E2 498.0107} C_DIS
LIN {X 88.6584,Y -109.6005,Z 185,A -46.3571,B 3.184,C 0.2979,E1 3.2992,E2 499.511} C_DIS
LIN {X 86.016,Y -111.6869,Z 185,A -48.0892,B 3.1834,C 0.3039,E1 3.2953,E2 501.2933} C_DIS
LIN {X 81.4837,Y -115.0352,Z 185,A -49.4995,B 3.1838,C 0.2996,E1 3.2923,E2 502.5861} C_DIS
LIN {X 78.8901,Y -116.8288,Z 185,A -51.3859,B 3.183,C 0.3074,E1 3.2878,E2 504.5557} C_DIS
LIN {X 75.0744,Y -119.3158,Z 185,A -52.8136,B 3.1831,C 0.3065,E1 3.2845,E2 505.9274} C_DIS
LIN {X 71.1104,Y -121.7211,Z 185,A -54.6381,B 3.1829,C 0.3089,E1 3.2802,E2 507.7451} C_DIS
LIN {X 67.1279,Y -123.9622,Z 185,A -56.4631,B 3.1826,C 0.3113,E1 3.2757,E2 509.5671} C_DIS
LIN {X 63.374,Y -125.9214,Z 185,A -58.0691,B 3.1826,C 0.3127,E1 3.2717,E2 511.1585} C_DIS
LIN {X 55.9855,Y -129.3742,Z 185,A -60.9888,B 3.1824,C 0.3135,E1 3.2645,E2 514.0266} C_DIS
LIN {X 52.2108,Y -130.9441,Z 185,A -62.9011,B 3.182,C 0.3178,E1 3.2594,E2 515.9745} C_DIS
LIN {X 48.5878,Y -132.3328,Z 185,A -64.7379,B 3.1816,C 0.3218,E1 3.2545,E2 517.8479} C_DIS
LIN {X 45.4754,Y -133.4339,Z 185,A -65.7619,B 3.1817,C 0.3205,E1 3.2519,E2 518.8293} C_DIS
LIN {X 42.7054,Y -134.3442,Z 185,A -66.9375,B 3.1817,C 0.3216,E1 3.2488,E2 520.0043} C_DIS
LIN {X 38.9851,Y -135.472,Z 185,A -68.7528,B 3.1813,C 0.3251,E1 3.2439,E2 521.8529} C_DIS
LIN {X 34.1994,Y -136.758,Z 185,A -70.4693,B 3.1813,C 0.3243,E1 3.2393,E2 523.5299} C_DIS
LIN {X 31.1461,Y -137.4849,Z 185,A -71.765,B 3.1813,C 0.3255,E1 3.2358,E2 524.8291} C_DIS
LIN {X 27.6685,Y -138.2273,Z 185,A -73.127,B 3.1812,C 0.3259,E1 3.2321,E2 526.1806} C_DIS
LIN {X 24.5141,Y -138.8211,Z 185,A -74.6807,B 3.1809,C 0.3288,E1 3.2277,E2 527.7692} C_DIS
LIN {X 17.3948,Y -139.8931,Z 185,A -77.3077,B 3.1809,C 0.328,E1 3.2206,E2 530.3569} C_DIS
LIN {X 13.6017,Y -140.311,Z 185,A -78.9357,B 3.1809,C 0.3293,E1 3.216,E2 531.9962} C_DIS
LIN {X 10.0705,Y -140.6087,Z 185,A -80.2893,B 3.1809,C 0.3292,E1 3.2122,E2 533.3388} C_DIS
LIN {X 6.8747,Y -140.8012,Z 185,A -81.6333,B 3.1808,C 0.3299,E1 3.2085,E2 534.6893} C_DIS
LIN {X 2.915,Y -140.9398,Z 185,A -83.3313,B 3.1807,C 0.331,E1 3.2037,E2 536.4001} C_DIS
LIN {X 2.915,Y -140.9398,Z 185,A -83.3313,B 3.1807,C 0.331,E1 3.2037,E2 536.4001} C_DIS
Enddeposition()
LIN {X 0.9991,Y -141.8653,Z 185,A -83.9895,B 3.1805,C 0.3319,E1 3.2018,E2 537.0732} C_DIS
Startdeposition()
$VEL.CP = VEL_PRINT
LIN {X 5.2916,Y -141.7704,Z 185,A -81.6587,B 3.181,C 0.3268,E1 3.2085,E2 534.6588} C_DIS
LIN {X 9.0105,Y -141.5827,Z 185,A -80.0543,B 3.1811,C 0.3255,E1 3.213,E2 533.0396} C_DIS
LIN {X 13.3991,Y -141.2348,Z 185,A -78.3904,B 3.1811,C 0.3257,E1 3.2176,E2 531.3907} C_DIS
LIN {X 17.8331,Y -140.7448,Z 185,A -76.4965,B 3.1813,C 0.3241,E1 3.2229,E2 529.4829} C_DIS
LIN {X 22.0358,Y -140.1473,Z 185,A -74.8786,B 3.1813,C 0.3239,E1 3.2273,E2 527.8775} C_DIS
LIN {X 26.0249,Y -139.4626,Z 185,A -73.2077,B 3.1815,C 0.3225,E1 3.2319,E2 526.2006} C_DIS
LIN {X 29.7833,Y -138.7072,Z 185,A -71.7093,B 3.1815,C 0.3218,E1 3.236,E2 524.7082} C_DIS
LIN {X 33.4677,Y -137.8647,Z 185,A -70.2242,B 3.1816,C 0.3209,E1 3.2401,E2 523.228} C_DIS
LIN {X 37.257,Y -136.891,Z 185,A -68.5996,B 3.1818,C 0.3192,E1 3.2445,E2 521.5962} C_DIS
LIN {X 41.1786,Y -135.7613,Z 185,A -67.0529,B 3.1818,C 0.3185,E1 3.2486,E2 520.0626} C_DIS
LIN {X 44.4363,Y -134.7303,Z 185,A -65.5823,B 3.1821,C 0.3163,E1 3.2525,E2 518.5783} C_DIS
LIN {X 48.0353,Y -133.4889,Z 185,A -64.1149,B 3.1821,C 0.3152,E1 3.2564,E2 517.1197} C_DIS
LIN {X 52.0208,Y -131.9884,Z 185,A -62.4688,B 3.1823,C 0.3139,E1 3.2606,E2 515.4827} C_DIS
LIN {X 56.5525,Y -130.1097,Z 185,A -60.1784,B 3.1828,C 0.3086,E1 3.2666,E2 513.1477} C_DIS
LIN {X 60.2163,Y -128.4569,Z 185,A -58.8251,B 3.1828,C 0.309,E1 3.27,E2 511.8311} C_DIS
LIN {X 63.7069,Y -126.762,Z 185,A -57.2121,B 3.183,C 0.3064,E1 3.274,E2 510.2106} C_DIS
LIN {X 68.0734,Y -124.4719,Z 185,A -55.4241,B 3.1831,C 0.3054,E1 3.2784,E2 508.4494} C_DIS
LIN {X 71.2078,Y -122.7057,Z 185,A -53.6024,B 3.1837,C 0.2997,E1 3.2829,E2 506.5753} C_DIS
LIN {X 74.9831,Y -120.4356,Z 185,A -51.5779,B 3.1842,C 0.2944,E1 3.2878,E2 504.5149} C_DIS
LIN {X 80.0908,Y -117.1014,Z 185,A -50.0122,B 3.1838,C 0.2989,E1 3.2911,E2 503.0727} C_DIS
LIN {X 82.2224,Y -115.6146,Z 185,A -48.639,B 3.1842,C 0.294,E1 3.2944,E2 501.6538} C_DIS
LIN {X 84.8726,Y -113.6833,Z 185,A -47.4618,B 3.1842,C 0.293,E1 3.297,E2 500.4961} C_DIS
LIN {X 88.7766,Y -110.6619,Z 185,A -45.5561,B 3.1846,C 0.2902,E1 3.3011,E2 498.601} C_DIS
LIN {X 92.2799,Y -107.758,Z 185,A -43.9992,B 3.1846,C 0.2894,E1 3.3044,E2 497.0816} C_DIS
LIN {X 96.0032,Y -104.4537,Z 185,A -41.6789,B 3.1853,C 0.2824,E1 3.3093,E2 494.7167} C_DIS
LIN {X 98.4312,Y -102.1696,Z 185,A -40.4968,B 3.1853,C 0.2813,E1 3.3116,E2 493.5564} C_DIS
LIN {X 101.9089,Y -98.7005,Z 185,A -38.6352,B 3.1856,C 0.2784,E1 3.3152,E2 491.7101} C_DIS
LIN {X 105.13,Y -95.2622,Z 185,A -36.0968,B 3.1865,C 0.2678,E1 3.3202,E2 489.0818} C_DIS
LIN {X 109.2703,Y -90.4832,Z 185,A -34.327,B 3.1863,C 0.2701,E1 3.3232,E2 487.4188} C_DIS
LIN {X 112.1557,Y -86.881,Z 185,A -32.7704,B 3.1864,C 0.269,E1 3.3258,E2 485.903} C_DIS
LIN {X 114.2267,Y -84.1398,Z 185,A -31.1953,B 3.1868,C 0.2639,E1 3.3285,E2 484.301} C_DIS
LIN {X 116.7326,Y -80.6281,Z 185,A -29.5089,B 3.1871,C 0.2603,E1 3.3312,E2 482.6208} C_DIS
LIN {X 119.1844,Y -76.9572,Z 185,A -27.7791,B 3.1874,C 0.2566,E1 3.3338,E2 480.8969} C_DIS
LIN {X 121.5849,Y -73.1057,Z 185,A -26.0176,B 3.1877,C 0.2528,E1 3.3364,E2 479.1437} C_DIS
LIN {X 123.9261,Y -69.0628,Z 185,A -24.0647,B 3.1882,C 0.2474,E1 3.3391,E2 477.1803} C_DIS
LIN {X 126.2564,Y -64.6999,Z 185,A -22.3963,B 3.1882,C 0.2458,E1 3.3412,E2 475.5553} C_DIS
LIN {X 127.8267,Y -61.5399,Z 185,A -21.1078,B 3.1885,C 0.2435,E1 3.3427,E2 474.2843} C_DIS
LIN {X 129.6867,Y -57.5169,Z 185,A -19.21,B 3.1889,C 0.2378,E1 3.3449,E2 472.3704} C_DIS
LIN {X 131.451,Y -53.361,Z 185,A -17.516,B 3.1892,C 0.2343,E1 3.3467,E2 470.6926} C_DIS
LIN {X 132.6287,Y -50.3658,Z 185,A -16.0664,B 3.1895,C 0.2293,E1 3.3482,E2 469.2215} C_DIS
LIN {X 134.7007,Y -44.525,Z 185,A -13.5327,B 3.19,C 0.2222,E1 3.3505,E2 466.6817} C_DIS
LIN {X 135.8935,Y -40.7465,Z 185,A -12.2309,B 3.19,C 0.2211,E1 3.3515,E2 465.4194} C_DIS
LIN {X 137.4507,Y -35.1294,Z 185,A -10.0961,B 3.1904,C 0.2169,E1 3.353,E2 463.3125} C_DIS
LIN {X 138.2551,Y -31.8164,Z 185,A -8.913,B 3.1904,C 0.2152,E1 3.3538,E2 462.1547} C_DIS
LIN {X 139.0405,Y -28.1865,Z 185,A -7.3103,B 3.1908,C 0.2099,E1 3.3547,E2 460.5369} C_DIS
LIN {X 139.7896,Y -24.2121,Z 185,A -5.6834,B 3.1911,C 0.2055,E1 3.3555,E2 458.9098} C_DIS
LIN {X 140.4203,Y -20.2217,Z 185,A -4.1896,B 3.1913,C 0.2024,E1 3.3561,E2 457.4333} C_DIS
LIN {X 140.9377,Y -16.2368,Z 185,A -2.5668,B 3.1916,C 0.1978,E1 3.3567,E2 455.8094} C_DIS
LIN {X 141.3107,Y -12.5889,Z 185,A -1.1533,B 3.1918,C 0.1944,E1 3.3571,E2 454.4041} C_DIS
LIN {X 141.5936,Y -8.835,Z 185,A 0.2751,B 3.192,C 0.1911,E1 3.3573,E2 452.9869} C_DIS
LIN {X 141.8056,Y -4.2498,Z 185,A 2.0183,B 3.1923,C 0.187,E1 3.3575,E2 451.2573} C_DIS
LIN {X 141.8677,Y -0.7877,Z 185,A 3.2999,B 3.1924,C 0.1843,E1 3.3575,E2 449.9904} C_DIS
LIN {X 141.8392,Y 2.9676,Z 185,A 4.8957,B 3.1927,C 0.1792,E1 3.3575,E2 448.3831} C_DIS
LIN {X 141.6813,Y 7.2956,Z 185,A 6.4987,B 3.1929,C 0.1758,E1 3.3573,E2 446.7985} C_DIS
LIN {X 141.3904,Y 11.6454,Z 185,A 8.1796,B 3.1931,C 0.1717,E1 3.3569,E2 445.1271} C_DIS
LIN {X 141.055,Y 15.174,Z 185,A 9.4576,B 3.1933,C 0.1693,E1 3.3566,E2 443.8687} C_DIS
LIN {X 140.641,Y 18.625,Z 185,A 10.8972,B 3.1935,C 0.165,E1 3.3561,E2 442.4235} C_DIS
LIN {X 139.978,Y 23.0858,Z 185,A 12.7871,B 3.1938,C 0.1592,E1 3.3553,E2 440.5234} C_DIS
LIN {X 138.8262,Y 29.2322,Z 185,A 15.1341,B 3.194,C 0.1541,E1 3.354,E2 438.1989} C_DIS
LIN {X 137.9182,Y 33.2457,Z 185,A 16.54,B 3.1941,C 0.1522,E1 3.3531,E2 436.826} C_DIS
LIN {X 137.1265,Y 36.3737,Z 185,A 17.7929,B 3.1943,C 0.1491,E1 3.3523,E2 435.579} C_DIS
LIN {X 136.4514,Y 38.8347,Z 185,A 19.0929,B 3.1945,C 0.1435,E1 3.3512,E2 434.2429} C_DIS
LIN {X 135.0131,Y 43.5697,Z 185,A 20.8325,B 3.1946,C 0.1408,E1 3.3498,E2 432.5366} C_DIS
LIN {X 133.6112,Y 47.696,Z 185,A 22.497,B 3.1948,C 0.1371,E1 3.3483,E2 430.8839} C_DIS
LIN {X 132.3253,Y 51.1541,Z 185,A 23.7756,B 3.1948,C 0.1354,E1 3.3471,E2 429.6324} C_DIS
LIN {X 131.0714,Y 54.2873,Z 185,A 25.183,B 3.195,C 0.1313,E1 3.3456,E2 428.2186} C_DIS
LIN {X 129.698,Y 57.4916,Z 185,A 26.5773,B 3.1952,C 0.1278,E1 3.344,E2 426.8255} C_DIS
LIN {X 128.1745,Y 60.8118,Z 185,A 28.0029,B 3.1953,C 0.1245,E1 3.3423,E2 425.4058} C_DIS
LIN {X 126.6872,Y 63.8538,Z 185,A 29.3515,B 3.1954,C 0.1212,E1 3.3407,E2 424.0592} C_DIS
LIN {X 124.7553,Y 67.5538,Z 185,A 31.0174,B 3.1956,C 0.1172,E1 3.3385,E2 422.3953} C_DIS
LIN {X 122.5431,Y 71.4884,Z 185,A 32.7519,B 3.1957,C 0.1136,E1 3.3361,E2 420.6718} C_DIS
LIN {X 120.2909,Y 75.2157,Z 185,A 34.4337,B 3.1958,C 0.1101,E1 3.3336,E2 418.9995} C_DIS
LIN {X 117.7853,Y 79.082,Z 185,A 36.2646,B 3.196,C 0.106,E1 3.3308,E2 417.1719} C_DIS
LIN {X 115.1915,Y 82.8147,Z 185,A 38.0254,B 3.1961,C 0.1024,E1 3.328,E2 415.4204} C_DIS
LIN {X 112.7754,Y 86.0751,Z 185,A 39.6323,B 3.1962,C 0.099,E1 3.3253,E2 413.8173} C_DIS
LIN {X 109.7057,Y 89.9551,Z 185,A 41.5293,B 3.1963,C 0.0955,E1 3.322,E2 411.933} C_DIS
LIN {X 106.7017,Y 93.4989,Z 185,A 43.345,B 3.1964,C 0.092,E1 3.3187,E2 410.1247} C_DIS
LIN {X 103.7331,Y 96.7816,Z 185,A 45.047,B 3.1965,C 0.089,E1 3.3155,E2 408.4334} C_DIS
LIN {X 100.5405,Y 100.0941,Z 185,A 46.8669,B 3.1965,C 0.0855,E1 3.3119,E2 406.6182} C_DIS
LIN {X 97.5109,Y 103.048,Z 185,A 48.6044,B 3.1967,C 0.0819,E1 3.3084,E2 404.8768} C_DIS
LIN {X 93.799,Y 106.4378,Z 185,A 50.4734,B 3.1967,C 0.0794,E1 3.3046,E2 403.0284} C_DIS
LIN {X 90.4541,Y 109.2944,Z 185,A 52.2249,B 3.1968,C 0.0763,E1 3.3008,E2 401.28} C_DIS
LIN {X 86.6986,Y 112.297,Z 185,A 54.1007,B 3.1968,C 0.0734,E1 3.2967,E2 399.4126} C_DIS
LIN {X 83.9366,Y 114.376,Z 185,A 55.4797,B 3.1969,C 0.0711,E1 3.2936,E2 398.0358} C_DIS
LIN {X 80.2456,Y 116.9951,Z 185,A 57.2118,B 3.1969,C 0.0689,E1 3.2897,E2 396.3159} C_DIS
LIN {X 76.7257,Y 119.3334,Z 185,A 58.9263,B 3.1971,C 0.0661,E1 3.2857,E2 394.6005} C_DIS
LIN {X 72.9411,Y 121.6837,Z 185,A 60.6975,B 3.1971,C 0.0636,E1 3.2815,E2 392.833} C_DIS
LIN {X 68.8277,Y 124.0564,Z 185,A 62.5318,B 3.1971,C 0.0615,E1 3.277,E2 391.0095} C_DIS
LIN {X 64.9149,Y 126.147,Z 185,A 64.1965,B 3.1971,C 0.0601,E1 3.273,E2 389.3611} C_DIS
LIN {X 61.7436,Y 127.7294,Z 185,A 65.6829,B 3.1972,C 0.0577,E1 3.2692,E2 387.8678} C_DIS
LIN {X 58.1609,Y 129.3987,Z 185,A 67.0897,B 3.1972,C 0.0573,E1 3.2657,E2 386.4854} C_DIS
LIN {X 55.5581,Y 130.5397,Z 185,A 68.3782,B 3.1972,C 0.0547,E1 3.2623,E2 385.1791} C_DIS
LIN {X 51.6476,Y 132.1334,Z 185,A 69.9062,B 3.1972,C 0.0542,E1 3.2584,E2 383.6739} C_DIS
LIN {X 48.4624,Y 133.3349,Z 185,A 71.1406,B 3.1972,C 0.0539,E1 3.2552,E2 382.4576} C_DIS
LIN {X 43.0343,Y 135.1841,Z 185,A 74.1438,B 3.1974,C 0.046,E1 3.247,E2 379.3672} C_DIS
LIN {X 38.3915,Y 136.5753,Z 185,A 75.4858,B 3.1974,C 0.0493,E1 3.2437,E2 378.1044} C_DIS
LIN {X 34.0946,Y 137.7132,Z 185,A 77.3964,B 3.1974,C 0.0469,E1 3.2384,E2 376.1796} C_DIS
LIN {X 30.1032,Y 138.6382,Z 185,A 78.9931,B 3.1974,C 0.0461,E1 3.2341,E2 374.5907} C_DIS
LIN {X 25.9827,Y 139.4707,Z 185,A 80.6085,B 3.1974,C 0.0457,E1 3.2297,E2 372.9863} C_DIS
LIN {X 22.2302,Y 140.1172,Z 185,A 82.2116,B 3.1974,C 0.0443,E1 3.2253,E2 371.3754} C_DIS
LIN {X 18.5464,Y 140.6513,Z 185,A 83.6319,B 3.1974,C 0.0442,E1 3.2213,E2 369.9661} C_DIS
LIN {X 14.6714,Y 141.1091,Z 185,A 85.2616,B 3.1974,C 0.0431,E1 3.2168,E2 368.3301} C_DIS
LIN {X 10.5013,Y 141.4798,Z 185,A 86.8719,B 3.1974,C 0.0431,E1 3.2123,E2 366.7306} C_DIS
LIN {X 6.5252,Y 141.72,Z 185,A 88.538,B 3.1974,C 0.0423,E1 3.2077,E2 365.058} C_DIS
LIN {X 2.3609,Y 141.8493,Z 185,A 90.1454,B 3.1974,C 0.0425,E1 3.2032,E2 363.4607} C_DIS
LIN {X -1.3592,Y 141.8636,Z 185,A 91.7846,B 3.1974,C 0.0414,E1 3.1986,E2 361.8049} C_DIS
LIN {X -5.7464,Y 141.7527,Z 185,A 93.3087,B 3.1974,C 0.0431,E1 3.1944,E2 360.313} C_DIS
LIN {X -9.4457,Y 141.5559,Z 185,A 95.0484,B 3.1974,C 0.0415,E1 3.1895,E2 358.5432} C_DIS
LIN {X -13.6875,Y 141.2071,Z 185,A 96.687,B 3.1974,C 0.0423,E1 3.1849,E2 356.9155} C_DIS
LIN {X -17.7531,Y 140.7553,Z 185,A 98.424,B 3.1974,C 0.042,E1 3.1801,E2 355.1687} C_DIS
LIN {X -22.472,Y 140.0797,Z 185,A 100.78,B 3.1974,C 0.0398,E1 3.1734,E2 352.7588} C_DIS
LIN {X -27.0276,Y 139.2709,Z 185,A 102.1615,B 3.1974,C 0.0438,E1 3.1698,E2 351.4403} C_DIS
LIN {X -31.3678,Y 138.3576,Z 185,A 103.8778,B 3.1974,C 0.0451,E1 3.1652,E2 349.7344} C_DIS
LIN {X -34.6108,Y 137.5823,Z 185,A 105.0821,B 3.1974,C 0.0468,E1 3.1619,E2 348.5489} C_DIS
LIN {X -39.1143,Y 136.3722,Z 185,A 107.2368,B 3.1974,C 0.0463,E1 3.156,E2 346.3611} C_DIS
LIN {X -42.5311,Y 135.3449,Z 185,A 108.7309,B 3.1974,C 0.047,E1 3.152,E2 344.861} C_DIS
LIN {X -46.2759,Y 134.1091,Z 185,A 110.763,B 3.1974,C 0.0455,E1 3.1465,E2 342.7738} C_DIS
LIN {X -50.6338,Y 132.5276,Z 185,A 112.1442,B 3.1974,C 0.0502,E1 3.1431,E2 341.4566} C_DIS
LIN {X -54.2646,Y 131.0809,Z 185,A 113.7369,B 3.1974,C 0.0517,E1 3.1389,E2 339.863} C_DIS
LIN {X -57.6784,Y 129.6145,Z 185,A 115.3022,B 3.1974,C 0.0528,E1 3.1349,E2 338.2904} C_DIS
LIN {X -60.967,Y 128.1004,Z 185,A 116.9969,B 3.1973,C 0.0531,E1 3.1305,E2 336.5671} C_DIS
LIN {X -65.6492,Y 125.7654,Z 185,A 118.9183,B 3.1973,C 0.0567,E1 3.1258,E2 334.6715} C_DIS
LIN {X -69.3166,Y 123.784,Z 185,A 120.5959,B 3.1972,C 0.0589,E1 3.1217,E2 332.9958} C_DIS
LIN {X -73.2647,Y 121.4888,Z 185,A 122.642,B 3.1972,C 0.0602,E1 3.1167,E2 330.9254} C_DIS
LIN {X -77.2651,Y 118.9845,Z 185,A 124.4971,B 3.1972,C 0.0632,E1 3.1124,E2 329.0781} C_DIS
LIN {X -80.7183,Y 116.6701,Z 185,A 126.2863,B 3.1971,C 0.0652,E1 3.1082,E2 327.276} C_DIS
LIN {X -84.3088,Y 114.1025,Z 185,A 128.0919,B 3.1971,C 0.0679,E1 3.1041,E2 325.4689} C_DIS
LIN {X -87.802,Y 111.4363,Z 185,A 129.9598,B 3.197,C 0.0703,E1 3.1,E2 323.5903} C_DIS
LIN {X -91.4296,Y 108.4801,Z 185,A 131.8847,B 3.1969,C 0.0734,E1 3.0958,E2 321.6624} C_DIS
LIN {X -94.0424,Y 106.2226,Z 185,A 133.3035,B 3.1969,C 0.0758,E1 3.0929,E2 320.2415} C_DIS
LIN {X -97.3134,Y 103.2342,Z 185,A 135.1322,B 3.1968,C 0.0789,E1 3.0891,E2 318.4091} C_DIS
LIN {X -100.2283,Y 100.4072,Z 185,A 136.8252,B 3.1967,C 0.0818,E1 3.0857,E2 316.7106} C_DIS
LIN {X -103.1429,Y 97.4102,Z 185,A 138.5099,B 3.1967,C 0.0852,E1 3.0825,E2 315.0276} C_DIS
LIN {X -106.1184,Y 94.1603,Z 185,A 140.4708,B 3.1965,C 0.0879,E1 3.0787,E2 313.0448} C_DIS
LIN {X -108.9994,Y 90.8104,Z 185,A 142.2037,B 3.1965,C 0.0919,E1 3.0756,E2 311.3199} C_DIS
LIN {X -111.5693,Y 87.6327,Z 185,A 143.9997,B 3.1963,C 0.0948,E1 3.0725,E2 309.5064} C_DIS
LIN {X -114.4911,Y 83.7799,Z 185,A 146.0325,B 3.1963,C 0.0988,E1 3.0691,E2 307.4648} C_DIS
LIN {X -116.7786,Y 80.561,Z 185,A 147.8359,B 3.1961,C 0.1014,E1 3.0662,E2 305.6357} C_DIS
LIN {X -119.7254,Y 76.1131,Z 185,A 149.9326,B 3.196,C 0.1067,E1 3.063,E2 303.5483} C_DIS
LIN {X -122.0452,Y 72.3346,Z 185,A 151.802,B 3.1958,C 0.1107,E1 3.0603,E2 301.67} C_DIS
LIN {X -124.3174,Y 68.3561,Z 185,A 153.6168,B 3.1957,C 0.1153,E1 3.0578,E2 299.8613} C_DIS
LIN {X -126.2173,Y 64.7768,Z 185,A 155.3598,B 3.1955,C 0.1189,E1 3.0555,E2 298.1057} C_DIS
LIN {X -127.8373,Y 61.5177,Z 185,A 156.8338,B 3.1954,C 0.1226,E1 3.0537,E2 296.6324} C_DIS
LIN {X -129.3264,Y 58.3225,Z 185,A 158.3639,B 3.1953,C 0.1257,E1 3.0519,E2 295.0895} C_DIS
LIN {X -130.7855,Y 54.9718,Z 185,A 159.7697,B 3.1951,C 0.1299,E1 3.0504,E2 293.6939} C_DIS
LIN {X -132.0734,Y 51.8021,Z 185,A 161.239,B 3.195,C 0.1331,E1 3.0489,E2 292.2144} C_DIS
LIN {X -133.3142,Y 48.5199,Z 185,A 162.763,B 3.1948,C 0.1364,E1 3.0474,E2 290.6775} C_DIS
LIN {X -134.4943,Y 45.1451,Z 185,A 164.3493,B 3.1947,C 0.1396,E1 3.0459,E2 289.0738} C_DIS
LIN {X -135.6037,Y 41.6937,Z 185,A 165.8313,B 3.1945,C 0.1434,E1 3.0447,E2 287.5905} C_DIS
LIN {X -136.5893,Y 38.3416,Z 185,A 167.3685,B 3.1944,C 0.1467,E1 3.0435,E2 286.0379} C_DIS
LIN {X -137.5805,Y 34.6177,Z 185,A 168.9883,B 3.1942,C 0.1507,E1 3.0423,E2 284.4109} C_DIS
LIN {X -138.3396,Y 31.4464,Z 185,A 171.1638,B 3.1942,C 0.1507,E1 3.041,E2 282.1229} C_DIS
LIN {X -139.5987,Y 25.2789,Z 185,A 172.9492,B 3.1937,C 0.1609,E1 3.0401,E2 280.4396} C_DIS
LIN {X -140.3359,Y 20.8123,Z 185,A 175.0085,B 3.1935,C 0.165,E1 3.0392,E2 278.3513} C_DIS
LIN {X -140.8399,Y 17.057,Z 185,A 176.515,B 3.1933,C 0.1694,E1 3.0386,E2 276.8489} C_DIS
LIN {X -141.2935,Y 12.7872,Z 185,A 178.3054,B 3.193,C 0.174,E1 3.0381,E2 275.0524} C_DIS
LIN {X -141.6411,Y 8.063,Z 185,A -179.5946,B 3.1928,C 0.1786,E1 3.0377,E2 272.929} C_DIS
LIN {X -141.8233,Y 3.6148,Z 185,A -177.7828,B 3.1925,C 0.1836,E1 3.0376,E2 271.1166} C_DIS
LIN {X -141.8711,Y 0.2029,Z 185,A -176.3938,B 3.1922,C 0.1875,E1 3.0376,E2 269.727} C_DIS
LIN {X -141.8383,Y -3.0226,Z 185,A -174.9637,B 3.1921,C 0.1906,E1 3.0376,E2 268.2808} C_DIS
LIN {X -141.7008,Y -6.9073,Z 185,A -173.1903,B 3.1918,C 0.1942,E1 3.0378,E2 266.4813} C_DIS
LIN {X -141.3607,Y -11.9971,Z 185,A -170.8473,B 3.1916,C 0.1987,E1 3.0384,E2 264.1018} C_DIS
LIN {X -140.9987,Y -15.6974,Z 185,A -169.5372,B 3.1912,C 0.2038,E1 3.0387,E2 262.8183} C_DIS
LIN {X -140.4621,Y -19.9289,Z 185,A -167.8363,B 3.1909,C 0.2086,E1 3.0394,E2 261.1213} C_DIS
LIN {X -139.9858,Y -23.0391,Z 185,A -166.5042,B 3.1907,C 0.2119,E1 3.04,E2 259.7818} C_DIS
LIN {X -138.8708,Y -29.0202,Z 185,A -163.7918,B 3.1903,C 0.2176,E1 3.0414,E2 257.0366} C_DIS
LIN {X -137.974,Y -33.0142,Z 185,A -162.187,B 3.19,C 0.2223,E1 3.0424,E2 255.4392} C_DIS
LIN {X -137.1349,Y -36.3423,Z 185,A -160.7401,B 3.1898,C 0.2258,E1 3.0435,E2 253.9849} C_DIS
LIN {X -136.1136,Y -39.9974,Z 185,A -159.1251,B 3.1895,C 0.2295,E1 3.0447,E2 252.3595} C_DIS
LIN {X -134.8637,Y -44.0356,Z 185,A -157.2159,B 3.1892,C 0.2332,E1 3.0464,E2 250.4241} C_DIS
LIN {X -133.8644,Y -46.9818,Z 185,A -156.0434,B 3.189,C 0.2369,E1 3.0474,E2 249.2634} C_DIS
LIN {X -132.5226,Y -50.6465,Z 185,A -154.3955,B 3.1887,C 0.2407,E1 3.049,E2 247.6067} C_DIS
LIN {X -131.0474,Y -54.3448,Z 185,A -152.6455,B 3.1884,C 0.2441,E1 3.0509,E2 245.8381} C_DIS
LIN {X -129.5575,Y -57.8059,Z 185,A -151.0324,B 3.1882,C 0.2476,E1 3.0527,E2 244.2132} C_DIS
LIN {X -127.4616,Y -62.2932,Z 185,A -149.0189,B 3.1878,C 0.2525,E1 3.0552,E2 242.1988} C_DIS
LIN {X -125.7838,Y -65.6142,Z 185,A -147.6833,B 3.1874,C 0.257,E1 3.0568,E2 240.8864} C_DIS
LIN {X -124.1727,Y -68.6175,Z 185,A -145.9774,B 3.1873,C 0.2588,E1 3.0592,E2 239.1363} C_DIS
LIN {X -121.9388,Y -72.5132,Z 185,A -144.1073,B 3.1869,C 0.2628,E1 3.0618,E2 237.2592} C_DIS
LIN {X -119.6171,Y -76.2825,Z 185,A -142.2088,B 3.1866,C 0.2665,E1 3.0646,E2 235.3462} C_DIS
LIN {X -117.0559,Y -80.1571,Z 185,A -140.2712,B 3.1863,C 0.2704,E1 3.0677,E2 233.4007} C_DIS
LIN {X -115.0438,Y -83.0194,Z 185,A -138.4397,B 3.1863,C 0.2714,E1 3.0708,E2 231.5122} C_DIS
LIN {X -112.4499,Y -86.5008,Z 185,A -137.004,B 3.1857,C 0.2769,E1 3.0731,E2 230.1206} C_DIS
LIN {X -109.6744,Y -89.9934,Z 185,A -135.1277,B 3.1854,C 0.2803,E1 3.0764,E2 228.2345} C_DIS
LIN {X -106.4016,Y -93.8399,Z 185,A -133.0269,B 3.1851,C 0.2841,E1 3.0803,E2 226.1257} C_DIS
LIN {X -103.6382,Y -96.8835,Z 185,A -131.3303,B 3.1848,C 0.2872,E1 3.0835,E2 224.4244} C_DIS
LIN {X -100.0758,Y -100.5587,Z 185,A -128.9341,B 3.1846,C 0.2894,E1 3.0883,E2 221.9832} C_DIS
LIN {X -97.4668,Y -103.0895,Z 185,A -127.6682,B 3.1843,C 0.2932,E1 3.0908,E2 220.7453} C_DIS
LIN {X -94.1342,Y -106.1415,Z 185,A -125.9731,B 3.1839,C 0.2972,E1 3.0943,E2 219.0683} C_DIS
LIN {X -91.3208,Y -108.5714,Z 185,A -124.24,B 3.1838,C 0.2985,E1 3.0981,E2 217.3034} C_DIS
LIN {X -87.6431,Y -111.5612,Z 185,A -122.4978,B 3.1834,C 0.3026,E1 3.1018,E2 215.5851} C_DIS
LIN {X -84.4165,Y -114.0228,Z 185,A -120.6411,B 3.1833,C 0.3039,E1 3.106,E2 213.6984} C_DIS
LIN {X -80.8593,Y -116.572,Z 185,A -118.7888,B 3.1831,C 0.3061,E1 3.1103,E2 211.8344} C_DIS
LIN {X -77.0981,Y -119.0929,Z 185,A -116.9156,B 3.1828,C 0.3084,E1 3.1147,E2 209.955} C_DIS
LIN {X -73.2781,Y -121.4807,Z 185,A -115.0655,B 3.1826,C 0.3107,E1 3.1191,E2 208.1005} C_DIS
LIN {X -69.2168,Y -123.8401,Z 185,A -113.0673,B 3.1825,C 0.3124,E1 3.124,E2 206.0881} C_DIS
LIN {X -65.031,Y -126.0879,Z 185,A -111.1712,B 3.1822,C 0.3148,E1 3.1287,E2 204.1949} C_DIS
LIN {X -61.6812,Y -127.7591,Z 185,A -109.6647,B 3.1821,C 0.3165,E1 3.1324,E2 202.689} C_DIS
LIN {X -58.3443,Y -129.3167,Z 185,A -108.2492,B 3.1819,C 0.3185,E1 3.136,E2 201.2833} C_DIS
LIN {X -54.9671,Y -130.7875,Z 185,A -106.6634,B 3.1818,C 0.3193,E1 3.1401,E2 199.6836} C_DIS
LIN {X -51.6418,Y -132.1357,Z 185,A -105.4568,B 3.1815,C 0.3222,E1 3.1432,E2 198.5104} C_DIS
LIN {X -46.7139,Y -133.9573,Z 185,A -102.2486,B 3.1821,C 0.3165,E1 3.152,E2 195.1499} C_DIS
LIN {X -40.5527,Y -135.951,Z 185,A -100.2031,B 3.1815,C 0.3222,E1 3.1573,E2 193.1839} C_DIS
LIN {X -35.6601,Y -137.316,Z 185,A -98.2743,B 3.1813,C 0.3243,E1 3.1624,E2 191.2717} C_DIS
LIN {X -32.2989,Y -138.1449,Z 185,A -96.8577,B 3.1813,C 0.3248,E1 3.1663,E2 189.852} C_DIS
LIN {X -28.2946,Y -139.0185,Z 185,A -95.3801,B 3.181,C 0.3268,E1 3.1703,E2 188.3985} C_DIS
LIN {X -24.9191,Y -139.6631,Z 185,A -93.9003,B 3.181,C 0.3266,E1 3.1744,E2 186.9055} C_DIS
LIN {X -21.1988,Y -140.2769,Z 185,A -92.2645,B 3.181,C 0.3262,E1 3.1789,E2 185.2535} C_DIS
LIN {X -17.2551,Y -140.8163,Z 185,A -90.734,B 3.181,C 0.3271,E1 3.1832,E2 183.7331} C_DIS
LIN {X -13.6781,Y -141.208,Z 185,A -89.2419,B 3.181,C 0.327,E1 3.1873,E2 182.235} C_DIS
LIN {X -9.2084,Y -141.5706,Z 185,A -87.4487,B 3.181,C 0.3272,E1 3.1923,E2 180.4435} C_DIS
LIN {X -5.1241,Y -141.7769,Z 185,A -85.7319,B 3.181,C 0.3266,E1 3.1971,E2 178.7168} C_DIS
LIN {X -0.7802,Y -141.8668,Z 185,A -84.0756,B 3.181,C 0.3272,E1 3.2017,E2 177.0735} C_DIS
LIN {X -0.7802,Y -141.8668,Z 185,A -84.0756,B 3.181,C 0.3272,E1 3.2017,E2 177.0735} C_DIS
Enddeposition()
LIN {X 1.005,Y -142.7647,Z 185,A -83.6736,B 3.1808,C 0.3313,E1 3.2029,E2 176.7462} C_DIS
Startdeposition()
$VEL.CP = VEL_PRINT
LIN {X -1.7477,Y -142.7598,Z 185,A -85.2217,B 3.1804,C 0.3349,E1 3.1984,E2 178.3567} C_DIS
LIN {X -6.1967,Y -142.636,Z 185,A -86.825,B 3.1806,C 0.3336,E1 3.194,E2 179.9354} C_DIS
LIN {X -9.6936,Y -142.4413,Z 185,A -88.2702,B 3.1806,C 0.3339,E1 3.19,E2 181.3867} C_DIS
LIN {X -13.194,Y -142.1588,Z 185,A -89.8031,B 3.1805,C 0.3347,E1 3.1856,E2 182.9373} C_DIS
LIN {X -17.4702,Y -141.6972,Z 185,A -91.3806,B 3.1805,C 0.3334,E1 3.1813,E2 184.495} C_DIS
LIN {X -20.9395,Y -141.227,Z 185,A -92.7914,B 3.1806,C 0.3331,E1 3.1774,E2 185.9071} C_DIS
LIN {X -24.3954,Y -140.6713,Z 185,A -94.2293,B 3.1806,C 0.3329,E1 3.1734,E2 187.3501} C_DIS
LIN {X -27.8522,Y -140.0271,Z 185,A -95.6394,B 3.1807,C 0.3324,E1 3.1695,E2 188.7605} C_DIS
LIN {X -31.2728,Y -139.3027,Z 185,A -97.0504,B 3.1807,C 0.3318,E1 3.1657,E2 190.173} C_DIS
LIN {X -34.6748,Y -138.4948,Z 185,A -98.4637,B 3.1808,C 0.3312,E1 3.1618,E2 191.5881} C_DIS
LIN {X -38.0566,Y -137.6037,Z 185,A -99.9761,B 3.1808,C 0.3312,E1 3.1577,E2 193.116} C_DIS
LIN {X -42.3408,Y -136.347,Z 185,A -101.6619,B 3.181,C 0.3292,E1 3.1532,E2 194.7876} C_DIS
LIN {X -45.5137,Y -135.3203,Z 185,A -103.042,B 3.1811,C 0.3285,E1 3.1496,E2 196.1738} C_DIS
LIN {X -48.9459,Y -134.1175,Z 185,A -104.6665,B 3.1811,C 0.3285,E1 3.1452,E2 197.8215} C_DIS
LIN {X -53.0074,Y -132.5641,Z 185,A -106.2895,B 3.1813,C 0.3261,E1 3.141,E2 199.4279} C_DIS
LIN {X -56.5325,Y -131.0991,Z 185,A -107.9376,B 3.1814,C 0.3254,E1 3.1368,E2 201.0923} C_DIS
LIN {X -60.2487,Y -129.4337,Z 185,A -109.4726,B 3.1817,C 0.3231,E1 3.1329,E2 202.6138} C_DIS
LIN {X -63.399,Y -127.9199,Z 185,A -110.9869,B 3.1817,C 0.3223,E1 3.129,E2 204.1437} C_DIS
LIN {X -66.9338,Y -126.1075,Z 185,A -112.5371,B 3.182,C 0.3202,E1 3.1252,E2 205.6881} C_DIS
LIN {X -70.3395,Y -124.2417,Z 185,A -114.2563,B 3.182,C 0.3192,E1 3.121,E2 207.4297} C_DIS
LIN {X -74.1482,Y -122.0065,Z 185,A -116.0506,B 3.1823,C 0.317,E1 3.1167,E2 209.2271} C_DIS
LIN {X -77.8588,Y -119.6723,Z 185,A -117.8135,B 3.1825,C 0.3146,E1 3.1125,E2 210.9905} C_DIS
LIN {X -81.4849,Y -117.2333,Z 185,A -119.6301,B 3.1827,C 0.3124,E1 3.1083,E2 212.8158} C_DIS
LIN {X -85.0359,Y -114.6839,Z 185,A -121.4424,B 3.183,C 0.3101,E1 3.1042,E2 214.636} C_DIS
LIN {X -88.5252,Y -112.013,Z 185,A -123.2607,B 3.1832,C 0.3075,E1 3.1001,E2 216.4618} C_DIS
LIN {X -91.9165,Y -109.2467,Z 185,A -125.0483,B 3.1835,C 0.3047,E1 3.0963,E2 218.2536} C_DIS
LIN {X -95.2283,Y -106.372,Z 185,A -126.8418,B 3.1837,C 0.3018,E1 3.0925,E2 220.0515} C_DIS
LIN {X -98.4351,Y -103.412,Z 185,A -128.6713,B 3.184,C 0.2991,E1 3.0888,E2 221.8915} C_DIS
LIN {X -101.5734,Y -100.3317,Z 185,A -130.4831,B 3.1843,C 0.296,E1 3.0852,E2 223.7096} C_DIS
LIN {X -104.5989,Y -97.1727,Z 185,A -132.0534,B 3.1847,C 0.2915,E1 3.0822,E2 225.2542} C_DIS
LIN {X -106.684,Y -94.8796,Z 185,A -133.5827,B 3.1847,C 0.2906,E1 3.0793,E2 226.8223} C_DIS
LIN {X -109.5488,Y -91.5563,Z 185,A -135.3849,B 3.1851,C 0.2871,E1 3.076,E2 228.6297} C_DIS
LIN {X -112.2513,Y -88.2218,Z 185,A -137.1759,B 3.1854,C 0.2838,E1 3.0729,E2 230.4296} C_DIS
LIN {X -114.8979,Y -84.7466,Z 185,A -138.989,B 3.1857,C 0.2803,E1 3.0698,E2 232.2505} C_DIS
LIN {X -117.4586,Y -81.1611,Z 185,A -140.8524,B 3.186,C 0.2768,E1 3.0668,E2 234.1264} C_DIS
LIN {X -119.9371,Y -77.451,Z 185,A -142.686,B 3.1863,C 0.2729,E1 3.064,E2 235.9652} C_DIS
LIN {X -122.2138,Y -73.8054,Z 185,A -144.4714,B 3.1867,C 0.2692,E1 3.0614,E2 237.7583} C_DIS
LIN {X -124.4156,Y -70.0301,Z 185,A -146.3012,B 3.187,C 0.2654,E1 3.0588,E2 239.5977} C_DIS
LIN {X -126.5068,Y -66.1735,Z 185,A -148.0672,B 3.1873,C 0.2611,E1 3.0565,E2 241.3637} C_DIS
LIN {X -128.3043,Y -62.6197,Z 185,A -149.7232,B 3.1876,C 0.2574,E1 3.0544,E2 243.0269} C_DIS
LIN {X -129.8086,Y -59.4379,Z 185,A -151.1929,B 3.1879,C 0.2541,E1 3.0527,E2 244.5038} C_DIS
LIN {X -131.5372,Y -55.5078,Z 185,A -153.0842,B 3.1882,C 0.2505,E1 3.0505,E2 246.417} C_DIS
LIN {X -133.1995,Y -51.3897,Z 185,A -154.8448,B 3.1886,C 0.2458,E1 3.0487,E2 248.1739} C_DIS
LIN {X -134.4171,Y -48.115,Z 185,A -156.3096,B 3.1888,C 0.2424,E1 3.0473,E2 249.6465} C_DIS
LIN {X -135.7249,Y -44.2988,Z 185,A -158.0851,B 3.1891,C 0.2388,E1 3.0457,E2 251.4422} C_DIS
LIN {X -136.8943,Y -40.5346,Z 185,A -159.6515,B 3.1894,C 0.2345,E1 3.0445,E2 253.0057} C_DIS
LIN {X -137.8471,Y -37.165,Z 185,A -161.0786,B 3.1897,C 0.2308,E1 3.0434,E2 254.435} C_DIS
LIN {X -138.8161,Y -33.3622,Z 185,A -162.8134,B 3.1899,C 0.2272,E1 3.0422,E2 256.1903} C_DIS
LIN {X -139.6315,Y -29.7677,Z 185,A -164.3275,B 3.1902,C 0.2233,E1 3.0413,E2 257.7083} C_DIS
LIN {X -140.364,Y -26.104,Z 185,A -165.8685,B 3.1905,C 0.2194,E1 3.0405,E2 259.2541} C_DIS
LIN {X -140.9606,Y -22.6662,Z 185,A -167.325,B 3.1907,C 0.2157,E1 3.0398,E2 260.7173} C_DIS
LIN {X -141.6097,Y -18.1613,Z 185,A -169.375,B 3.191,C 0.2116,E1 3.039,E2 262.7958} C_DIS
LIN {X -142.0794,Y -14.0202,Z 185,A -171.1484,B 3.1913,C 0.2074,E1 3.0385,E2 264.5816} C_DIS
LIN {X -142.4404,Y -9.7057,Z 185,A -172.8088,B 3.1916,C 0.2022,E1 3.0381,E2 266.2307} C_DIS
LIN {X -142.6358,Y -6.2,Z 185,A -174.3559,B 3.1918,C 0.1988,E1 3.0379,E2 267.7953} C_DIS
LIN {X -142.7597,Y -1.7578,Z 185,A -176.1091,B 3.1921,C 0.1936,E1 3.0379,E2 269.5433} C_DIS
LIN {X -142.76,Y 1.7385,Z 185,A -177.5483,B 3.1924,C 0.1898,E1 3.0379,E2 270.9863} C_DIS
LIN {X -142.6363,Y 6.1882,Z 185,A -179.4666,B 3.1926,C 0.1853,E1 3.038,E2 272.9209} C_DIS
LIN {X -142.4406,Y 9.7032,Z 185,A 178.9961,B 3.1928,C 0.1819,E1 3.0383,E2 274.4736} C_DIS
LIN {X -142.1593,Y 13.1885,Z 185,A 177.5343,B 3.193,C 0.1782,E1 3.0386,E2 275.9421} C_DIS
LIN {X -141.6988,Y 17.4566,Z 185,A 175.7521,B 3.1933,C 0.1736,E1 3.0392,E2 277.7309} C_DIS
LIN {X -141.2293,Y 20.9235,Z 185,A 174.2838,B 3.1935,C 0.17,E1 3.0398,E2 279.2066} C_DIS
LIN {X -140.5029,Y 25.3364,Z 185,A 172.397,B 3.1937,C 0.1654,E1 3.0407,E2 281.1041} C_DIS
LIN {X -139.7398,Y 29.2642,Z 185,A 170.636,B 3.1939,C 0.1616,E1 3.0416,E2 282.8844} C_DIS
LIN {X -138.9056,Y 32.9906,Z 185,A 169.106,B 3.1941,C 0.1574,E1 3.0426,E2 284.4129} C_DIS
LIN {X -138.0548,Y 36.3861,Z 185,A 167.6386,B 3.1943,C 0.1538,E1 3.0436,E2 285.8874} C_DIS
LIN {X -137.0346,Y 40.0552,Z 185,A 165.95,B 3.1945,C 0.1503,E1 3.0449,E2 287.5956} C_DIS
LIN {X -135.8113,Y 44.0292,Z 185,A 164.3093,B 3.1947,C 0.1457,E1 3.0463,E2 289.2315} C_DIS
LIN {X -134.7387,Y 47.208,Z 185,A 162.8816,B 3.1948,C 0.1425,E1 3.0476,E2 290.6687} C_DIS
LIN {X -133.49,Y 50.6326,Z 185,A 161.3747,B 3.195,C 0.1389,E1 3.0491,E2 292.1803} C_DIS
LIN {X -132.2632,Y 53.7539,Z 185,A 159.9465,B 3.1951,C 0.1357,E1 3.0506,E2 293.6181} C_DIS
LIN {X -130.8479,Y 57.1135,Z 185,A 158.4402,B 3.1953,C 0.1321,E1 3.0522,E2 295.1288} C_DIS
LIN {X -129.4413,Y 60.2324,Z 185,A 157.0026,B 3.1954,C 0.1289,E1 3.0539,E2 296.5737} C_DIS
LIN {X -127.9157,Y 63.4075,Z 185,A 155.4772,B 3.1955,C 0.1258,E1 3.0558,E2 298.1124} C_DIS
LIN {X -125.6811,Y 67.7328,Z 185,A 153.4343,B 3.1957,C 0.1214,E1 3.0585,E2 300.1654} C_DIS
LIN {X -123.5484,Y 71.5489,Z 185,A 151.6101,B 3.1958,C 0.1174,E1 3.061,E2 301.9971} C_DIS
LIN {X -121.3389,Y 75.2354,Z 185,A 149.7909,B 3.196,C 0.1138,E1 3.0637,E2 303.8272} C_DIS
LIN {X -118.9788,Y 78.9155,Z 185,A 147.9514,B 3.1961,C 0.1101,E1 3.0665,E2 305.6762} C_DIS
LIN {X -116.4514,Y 82.5993,Z 185,A 146.1262,B 3.1962,C 0.1061,E1 3.0694,E2 307.5041} C_DIS
LIN {X -114.0017,Y 85.948,Z 185,A 144.3698,B 3.1964,C 0.1028,E1 3.0723,E2 309.2709} C_DIS
LIN {X -111.1646,Y 89.5871,Z 185,A 142.4839,B 3.1964,C 0.099,E1 3.0756,E2 311.1598} C_DIS
LIN {X -108.3721,Y 92.9463,Z 185,A 140.6571,B 3.1966,C 0.0956,E1 3.0789,E2 312.9946} C_DIS
LIN {X -105.4771,Y 96.2194,Z 185,A 138.8399,B 3.1966,C 0.0923,E1 3.0823,E2 314.8186} C_DIS
LIN {X -102.5109,Y 99.3728,Z 185,A 137.0597,B 3.1968,C 0.0891,E1 3.0858,E2 316.6029} C_DIS
LIN {X -99.3678,Y 102.5158,Z 185,A 135.2198,B 3.1968,C 0.0859,E1 3.0894,E2 318.4486} C_DIS
LIN {X -96.2358,Y 105.4621,Z 185,A 133.4115,B 3.1969,C 0.0832,E1 3.0932,E2 320.2661} C_DIS
LIN {X -92.9424,Y 108.3754,Z 185,A 131.6053,B 3.1969,C 0.0802,E1 3.097,E2 322.0763} C_DIS
LIN {X -89.5801,Y 111.1703,Z 185,A 129.8198,B 3.1971,C 0.0774,E1 3.1008,E2 323.8644} C_DIS
LIN {X -86.1344,Y 113.861,Z 185,A 128.0037,B 3.1971,C 0.0748,E1 3.1049,E2 325.687} C_DIS
LIN {X -82.5963,Y 116.4535,Z 185,A 126.1846,B 3.1971,C 0.0723,E1 3.109,E2 327.5123} C_DIS
LIN {X -78.9188,Y 118.9766,Z 185,A 124.3638,B 3.1972,C 0.0698,E1 3.1132,E2 329.3358} C_DIS
LIN {X -75.2434,Y 121.3339,Z 185,A 122.5906,B 3.1972,C 0.0674,E1 3.1174,E2 331.1103} C_DIS
LIN {X -71.5606,Y 123.5416,Z 185,A 120.8169,B 3.1973,C 0.0654,E1 3.1217,E2 332.8893} C_DIS
LIN {X -67.7232,Y 125.6863,Z 185,A 118.9964,B 3.1973,C 0.0635,E1 3.1262,E2 334.7157} C_DIS
LIN {X -64.5579,Y 127.3389,Z 185,A 117.5816,B 3.1974,C 0.0616,E1 3.1297,E2 336.1272} C_DIS
LIN {X -60.6718,Y 129.2381,Z 185,A 115.7368,B 3.1974,C 0.0603,E1 3.1344,E2 337.9846} C_DIS
LIN {X -56.5724,Y 131.0818,Z 185,A 113.9829,B 3.1974,C 0.0582,E1 3.1389,E2 339.731} C_DIS
LIN {X -53.0346,Y 132.5531,Z 185,A 112.468,B 3.1975,C 0.0565,E1 3.1428,E2 341.2421} C_DIS
LIN {X -49.7768,Y 133.8105,Z 185,A 111.0467,B 3.1975,C 0.0554,E1 3.1465,E2 342.665} C_DIS
LIN {X -46.3152,Y 135.0482,Z 185,A 109.4424,B 3.1975,C 0.055,E1 3.1508,E2 344.2847} C_DIS
LIN {X -42.3541,Y 136.3429,Z 185,A 107.8173,B 3.1975,C 0.0534,E1 3.1551,E2 345.9029} C_DIS
LIN {X -38.8313,Y 137.387,Z 185,A 106.2264,B 3.1975,C 0.0532,E1 3.1594,E2 347.5074} C_DIS
LIN {X -34.6844,Y 138.4923,Z 185,A 104.6335,B 3.1975,C 0.0513,E1 3.1636,E2 349.0831} C_DIS
LIN {X -31.2945,Y 139.2977,Z 185,A 103.2251,B 3.1976,C 0.0506,E1 3.1675,E2 350.492} C_DIS
LIN {X -27.8824,Y 140.021,Z 185,A 101.8171,B 3.1976,C 0.05,E1 3.1713,E2 351.9003} C_DIS
LIN {X -24.4477,Y 140.6619,Z 185,A 100.4095,B 3.1976,C 0.0495,E1 3.1752,E2 353.3079} C_DIS
LIN {X -20.9929,Y 141.2194,Z 185,A 98.9587,B 3.1976,C 0.0495,E1 3.1792,E2 354.7639} C_DIS
LIN {X -17.4802,Y 141.696,Z 185,A 97.5483,B 3.1976,C 0.049,E1 3.1831,E2 356.172} C_DIS
LIN {X -14.0054,Y 142.0809,Z 185,A 96.0199,B 3.1976,C 0.0496,E1 3.1874,E2 357.7154} C_DIS
LIN {X -9.7133,Y 142.4399,Z 185,A 94.4368,B 3.1976,C 0.0484,E1 3.1918,E2 359.2794} C_DIS
LIN {X -6.2021,Y 142.6358,Z 185,A 92.9549,B 3.1976,C 0.0489,E1 3.196,E2 360.7695} C_DIS
LIN {X -1.7566,Y 142.7597,Z 185,A 91.2473,B 3.1976,C 0.0484,E1 3.2007,E2 362.4666} C_DIS
LIN {X 2.5464,Y 142.7465,Z 185,A 89.5087,B 3.1976,C 0.0487,E1 3.2056,E2 364.2059} C_DIS
LIN {X 6.1932,Y 142.6361,Z 185,A 88.0616,B 3.1976,C 0.0489,E1 3.2096,E2 365.6504} C_DIS
LIN {X 9.7016,Y 142.4407,Z 185,A 86.6221,B 3.1976,C 0.0496,E1 3.2136,E2 367.093} C_DIS
LIN {X 13.9868,Y 142.0827,Z 185,A 84.931,B 3.1976,C 0.0499,E1 3.2183,E2 368.7791} C_DIS
LIN {X 17.4652,Y 141.6978,Z 185,A 83.5392,B 3.1976,C 0.0504,E1 3.2222,E2 370.1688} C_DIS
LIN {X 20.9347,Y 141.2277,Z 185,A 82.1416,B 3.1976,C 0.0511,E1 3.226,E2 371.565} C_DIS
LIN {X 24.408,Y 140.669,Z 185,A 80.7258,B 3.1976,C 0.0519,E1 3.2299,E2 372.9809} C_DIS
LIN {X 27.8449,Y 140.0286,Z 185,A 79.3401,B 3.1976,C 0.0527,E1 3.2337,E2 374.364} C_DIS
LIN {X 31.2648,Y 139.3045,Z 185,A 77.9548,B 3.1976,C 0.0536,E1 3.2375,E2 375.7467} C_DIS
LIN {X 34.6668,Y 138.4968,Z 185,A 76.5699,B 3.1976,C 0.0545,E1 3.2413,E2 377.1289} C_DIS
LIN {X 38.0746,Y 137.5987,Z 185,A 75.0528,B 3.1976,C 0.0565,E1 3.2454,E2 378.6586} C_DIS
LIN {X 42.317,Y 136.3543,Z 185,A 73.4289,B 3.1975,C 0.0569,E1 3.2497,E2 380.2631} C_DIS
LIN {X 46.3667,Y 135.0304,Z 185,A 71.7458,B 3.1975,C 0.0584,E1 3.2542,E2 381.9425} C_DIS
LIN {X 49.738,Y 133.825,Z 185,A 70.3311,B 3.1975,C 0.0598,E1 3.2579,E2 383.3541} C_DIS
LIN {X 53.4008,Y 132.4056,Z 185,A 68.7113,B 3.1975,C 0.0619,E1 3.2621,E2 384.9792} C_DIS
LIN {X 57.1214,Y 130.8445,Z 185,A 67.1965,B 3.1974,C 0.063,E1 3.2659,E2 386.4805} C_DIS
LIN {X 60.242,Y 129.4368,Z 185,A 65.8442,B 3.1974,C 0.0645,E1 3.2694,E2 387.8298} C_DIS
LIN {X 63.3932,Y 127.9227,Z 185,A 64.4214,B 3.1974,C 0.0666,E1 3.273,E2 389.255} C_DIS
LIN {X 67.2856,Y 125.9214,Z 185,A 62.7074,B 3.1973,C 0.0687,E1 3.2772,E2 390.9636} C_DIS
LIN {X 71.1411,Y 123.7844,Z 185,A 60.9283,B 3.1973,C 0.0713,E1 3.2815,E2 392.7439} C_DIS
LIN {X 74.8986,Y 121.5472,Z 185,A 59.244,B 3.1972,C 0.0734,E1 3.2855,E2 394.4191} C_DIS
LIN {X 78.585,Y 119.1966,Z 185,A 57.5451,B 3.1972,C 0.0757,E1 3.2895,E2 396.1109} C_DIS
LIN {X 82.1133,Y 116.7942,Z 185,A 55.8346,B 3.197,C 0.0786,E1 3.2934,E2 397.821} C_DIS
LIN {X 85.628,Y 114.2431,Z 185,A 54.1256,B 3.197,C 0.0813,E1 3.2973,E2 399.5258} C_DIS
LIN {X 89.2085,Y 111.4694,Z 185,A 52.3903,B 3.197,C 0.0839,E1 3.301,E2 401.2506} C_DIS
LIN {X 92.59,Y 108.6763,Z 185,A 50.6884,B 3.1968,C 0.0866,E1 3.3047,E2 402.9452} C_DIS
LIN {X 95.8724,Y 105.7919,Z 185,A 48.9925,B 3.1968,C 0.0895,E1 3.3082,E2 404.6339} C_DIS
LIN {X 99.0806,Y 102.7938,Z 185,A 47.2674,B 3.1967,C 0.0927,E1 3.3117,E2 406.3544} C_DIS
LIN {X 102.1839,Y 99.7096,Z 185,A 45.5749,B 3.1966,C 0.0957,E1 3.315,E2 408.0391} C_DIS
LIN {X 105.1908,Y 96.5315,Z 185,A 43.8785,B 3.1965,C 0.0988,E1 3.3182,E2 409.7282} C_DIS
LIN {X 108.1067,Y 93.2544,Z 185,A 42.1715,B 3.1964,C 0.1021,E1 3.3213,E2 411.4286} C_DIS
LIN {X 110.9112,Y 89.9013,Z 185,A 40.4749,B 3.1963,C 0.1054,E1 3.3243,E2 413.1182} C_DIS
LIN {X 113.612,Y 86.463,Z 185,A 38.7824,B 3.1962,C 0.1088,E1 3.3272,E2 414.803} C_DIS
LIN {X 116.1313,Y 83.0479,Z 185,A 37.1345,B 3.196,C 0.1122,E1 3.3299,E2 416.4443} C_DIS
LIN {X 118.7126,Y 79.3142,Z 185,A 35.3877,B 3.196,C 0.1158,E1 3.3327,E2 418.1819} C_DIS
LIN {X 121.0865,Y 75.6409,Z 185,A 33.6961,B 3.1958,C 0.1194,E1 3.3352,E2 419.8659} C_DIS
LIN {X 123.3472,Y 71.8963,Z 185,A 31.9968,B 3.1956,C 0.1231,E1 3.3376,E2 421.5584} C_DIS
LIN {X 125.4916,Y 68.0838,Z 185,A 30.2663,B 3.1955,C 0.1272,E1 3.3399,E2 423.2863} C_DIS
LIN {X 127.3502,Y 64.5357,Z 185,A 28.7999,B 3.1954,C 0.1299,E1 3.3418,E2 424.7348} C_DIS
LIN {X 129.066,Y 61.0339,Z 185,A 27.3349,B 3.1952,C 0.1329,E1 3.3435,E2 426.1874} C_DIS
LIN {X 130.8452,Y 57.1196,Z 185,A 25.5858,B 3.195,C 0.1376,E1 3.3455,E2 427.9404} C_DIS
LIN {X 132.5601,Y 53.0175,Z 185,A 23.9668,B 3.195,C 0.1405,E1 3.3472,E2 429.5384} C_DIS
LIN {X 133.8192,Y 49.7537,Z 185,A 22.595,B 3.1948,C 0.1439,E1 3.3486,E2 430.9067} C_DIS
LIN {X 135.3104,Y 45.5433,Z 185,A 20.9412,B 3.1946,C 0.1473,E1 3.3501,E2 432.5431} C_DIS
LIN {X 136.344,Y 42.3506,Z 185,A 19.5647,B 3.1944,C 0.1512,E1 3.3512,E2 433.9242} C_DIS
LIN {X 137.385,Y 38.8387,Z 185,A 18.1982,B 3.1943,C 0.1542,E1 3.3523,E2 435.2778} C_DIS
LIN {X 138.258,Y 35.6077,Z 185,A 16.8108,B 3.1941,C 0.1583,E1 3.3533,E2 436.6717} C_DIS
LIN {X 139.2971,Y 31.2971,Z 185,A 15.211,B 3.1939,C 0.1613,E1 3.3543,E2 438.2487} C_DIS
LIN {X 140.0212,Y 27.8813,Z 185,A 13.8702,B 3.1938,C 0.1645,E1 3.355,E2 439.5824} C_DIS
LIN {X 140.6626,Y 24.4439,Z 185,A 12.527,B 3.1936,C 0.1678,E1 3.3557,E2 440.9184} C_DIS
LIN {X 141.2257,Y 20.9484,Z 185,A 11.1455,B 3.1934,C 0.1714,E1 3.3563,E2 442.2955} C_DIS
LIN {X 141.67,Y 17.6982,Z 185,A 9.8254,B 3.1932,C 0.1751,E1 3.3568,E2 443.6169} C_DIS
LIN {X 142.0819,Y 13.9948,Z 185,A 8.3417,B 3.193,C 0.1792,E1 3.3572,E2 445.1} C_DIS
LIN {X 142.441,Y 9.6984,Z 185,A 6.8206,B 3.1928,C 0.1818,E1 3.3575,E2 446.5944} C_DIS
LIN {X 142.6357,Y 6.2025,Z 185,A 5.4118,B 3.1926,C 0.1858,E1 3.3577,E2 448.0045} C_DIS
LIN {X 142.7501,Y 2.3343,Z 185,A 3.9473,B 3.1924,C 0.1893,E1 3.3578,E2 449.4582} C_DIS
Enddeposition()
END
